(* Visualisation DALI 647/Configuration Pages/visuDALIGroups
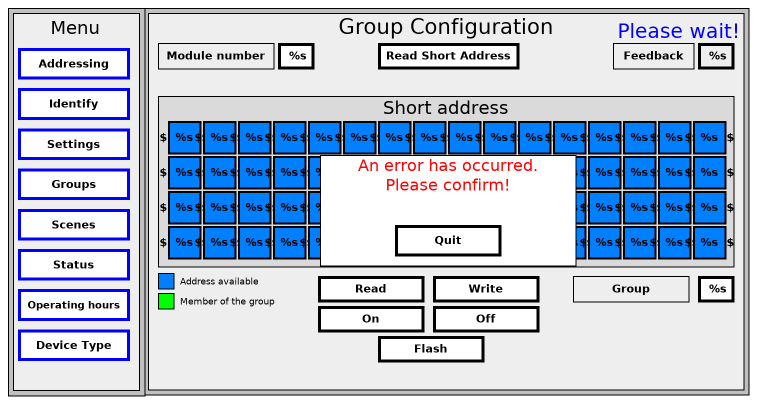
rectangle at (140,5)-(736,382): text "Group Configuration"
rectangle at (150,88)-(726,259): text "Short address"
embedded screen at (160,113)-(193,146): visuGroupButton
embedded screen at (160,148)-(193,181): visuGroupButton
embedded screen at (160,183)-(193,216): visuGroupButton
embedded screen at (160,218)-(193,251): visuGroupButton
embedded screen at (195,113)-(228,146): visuGroupButton
embedded screen at (195,148)-(228,181): visuGroupButton
embedded screen at (195,183)-(228,216): visuGroupButton
embedded screen at (195,218)-(228,251): visuGroupButton
embedded screen at (230,113)-(263,146): visuGroupButton
embedded screen at (230,148)-(263,181): visuGroupButton
embedded screen at (230,183)-(263,216): visuGroupButton
embedded screen at (230,218)-(263,251): visuGroupButton
embedded screen at (265,113)-(298,146): visuGroupButton
embedded screen at (265,148)-(298,181): visuGroupButton
embedded screen at (265,183)-(298,216): visuGroupButton
embedded screen at (265,218)-(298,251): visuGroupButton
embedded screen at (300,113)-(333,146): visuGroupButton
embedded screen at (300,148)-(333,181): visuGroupButton
embedded screen at (300,183)-(333,216): visuGroupButton
embedded screen at (300,218)-(333,251): visuGroupButton
embedded screen at (335,113)-(368,146): visuGroupButton
embedded screen at (335,148)-(368,181): visuGroupButton
embedded screen at (335,183)-(368,216): visuGroupButton
embedded screen at (335,218)-(368,251): visuGroupButton
embedded screen at (370,113)-(403,146): visuGroupButton
embedded screen at (370,148)-(403,181): visuGroupButton
embedded screen at (370,183)-(403,216): visuGroupButton
embedded screen at (370,218)-(403,251): visuGroupButton
embedded screen at (405,113)-(438,146): visuGroupButton
embedded screen at (405,148)-(438,181): visuGroupButton
embedded screen at (405,183)-(438,216): visuGroupButton
embedded screen at (405,218)-(438,251): visuGroupButton
embedded screen at (440,113)-(473,146): visuGroupButton
embedded screen at (440,148)-(473,181): visuGroupButton
embedded screen at (440,183)-(473,216): visuGroupButton
embedded screen at (440,218)-(473,251): visuGroupButton
embedded screen at (475,113)-(508,146): visuGroupButton
embedded screen at (475,148)-(508,181): visuGroupButton
embedded screen at (475,183)-(508,216): visuGroupButton
embedded screen at (475,218)-(508,251): visuGroupButton
embedded screen at (510,113)-(543,146): visuGroupButton
embedded screen at (510,148)-(543,181): visuGroupButton
embedded screen at (510,183)-(543,216): visuGroupButton
embedded screen at (510,218)-(543,251): visuGroupButton
embedded screen at (545,113)-(578,146): visuGroupButton
embedded screen at (545,148)-(578,181): visuGroupButton
embedded screen at (545,183)-(578,216): visuGroupButton
embedded screen at (545,218)-(578,251): visuGroupButton
embedded screen at (580,113)-(613,146): visuGroupButton
embedded screen at (580,148)-(613,181): visuGroupButton
embedded screen at (580,183)-(613,216): visuGroupButton
embedded screen at (580,218)-(613,251): visuGroupButton
embedded screen at (615,113)-(648,146): visuGroupButton
embedded screen at (615,148)-(648,181): visuGroupButton
embedded screen at (615,183)-(648,216): visuGroupButton
embedded screen at (615,218)-(648,251): visuGroupButton
embedded screen at (650,113)-(683,146): visuGroupButton
embedded screen at (650,148)-(683,181): visuGroupButton
embedded screen at (650,183)-(683,216): visuGroupButton
embedded screen at (650,218)-(683,251): visuGroupButton
embedded screen at (685,113)-(718,146): visuGroupButton
embedded screen at (685,148)-(718,181): visuGroupButton
embedded screen at (685,183)-(718,216): visuGroupButton
embedded screen at (685,218)-(718,251): visuGroupButton
rounded rectangle at (150,35)-(266,61): text "Module number"
rounded rectangle at (270,35)-(306,61): text "%s"; shows PrgDALIConfig.bModule_753_647; editable
rounded rectangle at (565,268)-(681,294): text "Group"
rounded rectangle at (690,268)-(726,294): text "%s"; shows PrgDALIConfig.GroupConfig.bGroup; editable
rounded rectangle at (310,268)-(416,294): text "Read"; alarm colour if PrgDALIConfig.GroupConfig.xRead; taps PrgDALIConfig.GroupConfig.xRead
rounded rectangle at (425,268)-(531,294): text "Write"; alarm colour if PrgDALIConfig.GroupConfig.xWrite; taps PrgDALIConfig.GroupConfig.xWrite
rectangle at (170,283)-(300,304): text "Member of the group"
rectangle at (170,263)-(300,284): text "Address available"
rounded rectangle at (370,328)-(476,354): text "Flash"; alarm colour if PrgDALIConfig.GroupConfig.xFlash; toggles PrgDALIConfig.GroupConfig.xFlash
rounded rectangle at (425,298)-(531,324): text "Off"; alarm colour if PrgDALIConfig.GroupConfig.xGroupOff; taps PrgDALIConfig.GroupConfig.xGroupOff
rounded rectangle at (310,298)-(416,324): text "On"; alarm colour if PrgDALIConfig.GroupConfig.xGroupOn; taps PrgDALIConfig.GroupConfig.xGroupOn
rounded rectangle at (605,35)-(686,61): text "Feedback"
rounded rectangle at (690,35)-(726,61): text "%s"; shows PrgDALIConfig.GroupConfig.bFeedback
rounded rectangle at (370,35)-(511,61): text "Read Short Address"; alarm colour if PrgDALIConfig.GroupConfig.xQueryShortAddress; taps PrgDALIConfig.GroupConfig.xQueryShortAddress
embedded screen at (0,0)-(137,388): visuDALI_Menue
group at (0,7)-(734,379)
  rectangle at (3,3)-(734,321): text "Please wait!"
group at (312,147)-(568,258)
  rectangle at (0,0)-(256,111): text "An error has occurred. / Please confirm!"
  rounded rectangle at (75,70)-(181,101): text "Quit"; taps PrgDALIConfig.GroupConfig.xQuit
4 more shapes without text or variables
*)

(* Visualisation DALI 647/Configuration Pages/visuDALIOperatingHours
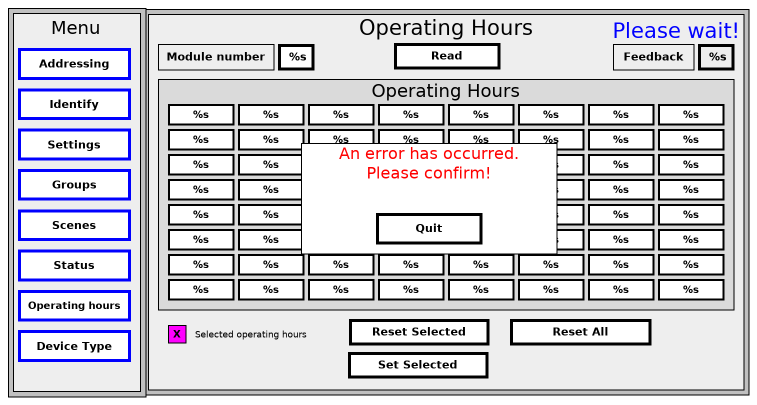
rectangle at (140,6)-(736,382): text "Operating Hours"
rectangle at (150,71)-(726,302): text "Operating Hours"
rectangle at (160,317)-(178,335): text "X"
rounded rectangle at (150,36)-(266,62): text "Module number"
rounded rectangle at (270,36)-(306,62): text "%s"; shows PrgDALIConfig.bModule_753_647; editable
rounded rectangle at (341,311)-(481,337): text "Reset Selected"; alarm colour if PrgDALIConfig.OperatingHours.xResetSelected; taps PrgDALIConfig.OperatingHours.xResetSelected
rectangle at (185,316)-(315,337): text "Selected operating hours"
rounded rectangle at (605,36)-(686,62): text "Feedback"
rounded rectangle at (690,36)-(726,62): text "%s"; shows PrgDALIConfig.OperatingHours.bFeedback
rounded rectangle at (502,311)-(643,337): text "Reset All"; alarm colour if PrgDALIConfig.OperatingHours.xResetAll; taps PrgDALIConfig.OperatingHours.xResetAll
rounded rectangle at (340,344)-(480,370): text "Set Selected"; invisible if PrgDALIConfig.OperatingHours.OldFirmware; alarm colour if PrgDALIConfig.OperatingHours.xSetSelected; taps PrgDALIConfig.OperatingHours.xSetSelected
embedded screen at (160,96)-(226,117): visuOperatingHours
embedded screen at (230,96)-(296,117): visuOperatingHours
embedded screen at (300,96)-(366,117): visuOperatingHours
embedded screen at (370,96)-(436,117): visuOperatingHours
embedded screen at (440,96)-(506,117): visuOperatingHours
embedded screen at (510,96)-(576,117): visuOperatingHours
embedded screen at (580,96)-(646,117): visuOperatingHours
embedded screen at (650,96)-(716,117): visuOperatingHours
embedded screen at (160,121)-(226,142): visuOperatingHours
embedded screen at (230,121)-(296,142): visuOperatingHours
embedded screen at (300,121)-(366,142): visuOperatingHours
embedded screen at (370,121)-(436,142): visuOperatingHours
embedded screen at (440,121)-(506,142): visuOperatingHours
embedded screen at (510,121)-(576,142): visuOperatingHours
embedded screen at (580,121)-(646,142): visuOperatingHours
embedded screen at (650,121)-(716,142): visuOperatingHours
embedded screen at (160,146)-(226,167): visuOperatingHours
embedded screen at (230,146)-(296,167): visuOperatingHours
embedded screen at (300,146)-(366,167): visuOperatingHours
embedded screen at (370,146)-(436,167): visuOperatingHours
embedded screen at (440,146)-(506,167): visuOperatingHours
embedded screen at (510,146)-(576,167): visuOperatingHours
embedded screen at (580,146)-(646,167): visuOperatingHours
embedded screen at (650,146)-(716,167): visuOperatingHours
embedded screen at (160,171)-(226,192): visuOperatingHours
embedded screen at (230,171)-(296,192): visuOperatingHours
embedded screen at (300,171)-(366,192): visuOperatingHours
embedded screen at (370,171)-(436,192): visuOperatingHours
embedded screen at (440,171)-(506,192): visuOperatingHours
embedded screen at (510,171)-(576,192): visuOperatingHours
embedded screen at (580,171)-(646,192): visuOperatingHours
embedded screen at (650,171)-(716,192): visuOperatingHours
embedded screen at (160,196)-(226,217): visuOperatingHours
embedded screen at (230,196)-(296,217): visuOperatingHours
embedded screen at (300,196)-(366,217): visuOperatingHours
embedded screen at (370,196)-(436,217): visuOperatingHours
embedded screen at (440,196)-(506,217): visuOperatingHours
embedded screen at (510,196)-(576,217): visuOperatingHours
embedded screen at (580,196)-(646,217): visuOperatingHours
embedded screen at (650,196)-(716,217): visuOperatingHours
embedded screen at (160,221)-(226,242): visuOperatingHours
embedded screen at (230,221)-(296,242): visuOperatingHours
embedded screen at (300,221)-(366,242): visuOperatingHours
embedded screen at (370,221)-(436,242): visuOperatingHours
embedded screen at (440,221)-(506,242): visuOperatingHours
embedded screen at (510,221)-(576,242): visuOperatingHours
embedded screen at (580,221)-(646,242): visuOperatingHours
embedded screen at (650,221)-(716,242): visuOperatingHours
embedded screen at (160,246)-(226,267): visuOperatingHours
embedded screen at (230,246)-(296,267): visuOperatingHours
embedded screen at (300,246)-(366,267): visuOperatingHours
embedded screen at (370,246)-(436,267): visuOperatingHours
embedded screen at (440,246)-(506,267): visuOperatingHours
embedded screen at (510,246)-(576,267): visuOperatingHours
embedded screen at (580,246)-(646,267): visuOperatingHours
embedded screen at (650,246)-(716,267): visuOperatingHours
embedded screen at (160,271)-(226,292): visuOperatingHours
embedded screen at (230,271)-(296,292): visuOperatingHours
embedded screen at (300,271)-(366,292): visuOperatingHours
embedded screen at (370,271)-(436,292): visuOperatingHours
embedded screen at (440,271)-(506,292): visuOperatingHours
embedded screen at (510,271)-(576,292): visuOperatingHours
embedded screen at (580,271)-(646,292): visuOperatingHours
embedded screen at (650,271)-(716,292): visuOperatingHours
rounded rectangle at (386,35)-(492,61): text "Read"; alarm colour if PrgDALIConfig.OperatingHours.xEnable; taps PrgDALIConfig.OperatingHours.xEnable
embedded screen at (0,0)-(138,389): visuDALI_Menue
rectangle at (3,9)-(734,383): text "Please wait!"; invisible if PrgDALIConfig.OperatingHours.xReady
group at (293,135)-(549,246)
  rectangle at (0,0)-(256,111): text "An error has occurred. / Please confirm!"
  rounded rectangle at (75,70)-(181,101): text "Quit"; taps PrgDALIConfig.OperatingHours.xQuit
1 more shapes without text or variables
*)

(* Visualisation DALI 647/Configuration Pages/visuDALIScenes
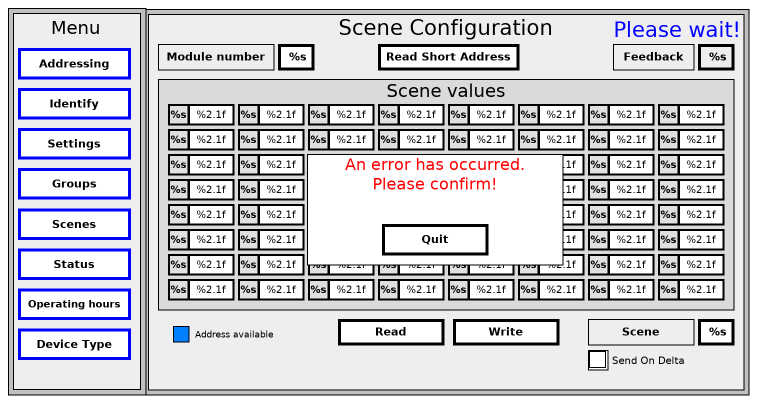
rectangle at (140,6)-(736,382): text "Scene Configuration"
rectangle at (150,71)-(726,302): text "Scene values"
rounded rectangle at (150,36)-(266,62): text "Module number"
rounded rectangle at (270,36)-(306,62): text "%s"; shows PrgDALIConfig.bModule_753_647; editable
rounded rectangle at (330,311)-(436,337): text "Read"; alarm colour if PrgDALIConfig.SceneConfig.xRead; taps PrgDALIConfig.SceneConfig.xRead
rounded rectangle at (445,311)-(551,337): text "Write"; alarm colour if PrgDALIConfig.SceneConfig.xWrite; taps PrgDALIConfig.SceneConfig.xWrite
rectangle at (185,316)-(281,337): text "Address available"
rounded rectangle at (605,36)-(686,62): text "Feedback"
rounded rectangle at (690,36)-(726,62): text "%s"; shows PrgDALIConfig.SceneConfig.bFeedback
rounded rectangle at (370,36)-(511,62): text "Read Short Address"; alarm colour if PrgDALIConfig.SceneConfig.xQueryShortAddress; taps PrgDALIConfig.SceneConfig.xQueryShortAddress
embedded screen at (580,342)-(600,362): visuDaliSelect
embedded screen at (160,96)-(226,117): visuSceneValues
embedded screen at (230,96)-(296,117): visuSceneValues
embedded screen at (300,96)-(366,117): visuSceneValues
embedded screen at (370,96)-(436,117): visuSceneValues
embedded screen at (440,96)-(506,117): visuSceneValues
embedded screen at (510,96)-(576,117): visuSceneValues
embedded screen at (580,96)-(646,117): visuSceneValues
embedded screen at (650,96)-(716,117): visuSceneValues
embedded screen at (160,121)-(226,142): visuSceneValues
embedded screen at (230,121)-(296,142): visuSceneValues
embedded screen at (300,121)-(366,142): visuSceneValues
embedded screen at (370,121)-(436,142): visuSceneValues
embedded screen at (440,121)-(506,142): visuSceneValues
embedded screen at (510,121)-(576,142): visuSceneValues
embedded screen at (580,121)-(646,142): visuSceneValues
embedded screen at (650,121)-(716,142): visuSceneValues
embedded screen at (160,146)-(226,167): visuSceneValues
embedded screen at (230,146)-(296,167): visuSceneValues
embedded screen at (300,146)-(366,167): visuSceneValues
embedded screen at (370,146)-(436,167): visuSceneValues
embedded screen at (440,146)-(506,167): visuSceneValues
embedded screen at (510,146)-(576,167): visuSceneValues
embedded screen at (580,146)-(646,167): visuSceneValues
embedded screen at (650,146)-(716,167): visuSceneValues
embedded screen at (160,171)-(226,192): visuSceneValues
embedded screen at (230,171)-(296,192): visuSceneValues
embedded screen at (300,171)-(366,192): visuSceneValues
embedded screen at (370,171)-(436,192): visuSceneValues
embedded screen at (440,171)-(506,192): visuSceneValues
embedded screen at (510,171)-(576,192): visuSceneValues
embedded screen at (580,171)-(646,192): visuSceneValues
embedded screen at (650,171)-(716,192): visuSceneValues
embedded screen at (160,196)-(226,217): visuSceneValues
embedded screen at (230,196)-(296,217): visuSceneValues
embedded screen at (300,196)-(366,217): visuSceneValues
embedded screen at (370,196)-(436,217): visuSceneValues
embedded screen at (440,196)-(506,217): visuSceneValues
embedded screen at (510,196)-(576,217): visuSceneValues
embedded screen at (580,196)-(646,217): visuSceneValues
embedded screen at (650,196)-(716,217): visuSceneValues
embedded screen at (160,221)-(226,242): visuSceneValues
embedded screen at (230,221)-(296,242): visuSceneValues
embedded screen at (300,221)-(366,242): visuSceneValues
embedded screen at (370,221)-(436,242): visuSceneValues
embedded screen at (440,221)-(506,242): visuSceneValues
embedded screen at (510,221)-(576,242): visuSceneValues
embedded screen at (580,221)-(646,242): visuSceneValues
embedded screen at (650,221)-(716,242): visuSceneValues
embedded screen at (160,246)-(226,267): visuSceneValues
embedded screen at (230,246)-(296,267): visuSceneValues
embedded screen at (300,246)-(366,267): visuSceneValues
embedded screen at (370,246)-(436,267): visuSceneValues
embedded screen at (440,246)-(506,267): visuSceneValues
embedded screen at (510,246)-(576,267): visuSceneValues
embedded screen at (580,246)-(646,267): visuSceneValues
embedded screen at (650,246)-(716,267): visuSceneValues
embedded screen at (160,271)-(226,292): visuSceneValues
embedded screen at (230,271)-(296,292): visuSceneValues
embedded screen at (300,271)-(366,292): visuSceneValues
embedded screen at (370,271)-(436,292): visuSceneValues
embedded screen at (440,271)-(506,292): visuSceneValues
embedded screen at (510,271)-(576,292): visuSceneValues
embedded screen at (580,271)-(646,292): visuSceneValues
embedded screen at (650,271)-(716,292): visuSceneValues
rounded rectangle at (580,311)-(686,337): text "Scene"
rounded rectangle at (690,311)-(726,337): text "%s"; shows PrgDALIConfig.SceneConfig.bScene; editable
embedded screen at (0,0)-(138,387): visuDALI_Menue
rectangle at (4,8)-(735,381): text "Please wait!"; invisible if PrgDALIConfig.SceneConfig.xReady
group at (299,146)-(555,257)
  rectangle at (0,0)-(256,111): text "An error has occurred. / Please confirm!"
  rounded rectangle at (75,70)-(181,101): text "Quit"; taps PrgDALIConfig.SceneConfig.xQuit
rectangle at (602,341)-(690,364): text "Send On Delta"
2 more shapes without text or variables
*)

(* Visualisation DALI 647/Private/visuDaliSelect
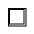
rectangle at (1,1)-(16,16): invisible if $Select$; toggles $Select$
2 more shapes without text or variables
*)

(* Visualisation Private/English/visuECG_settings
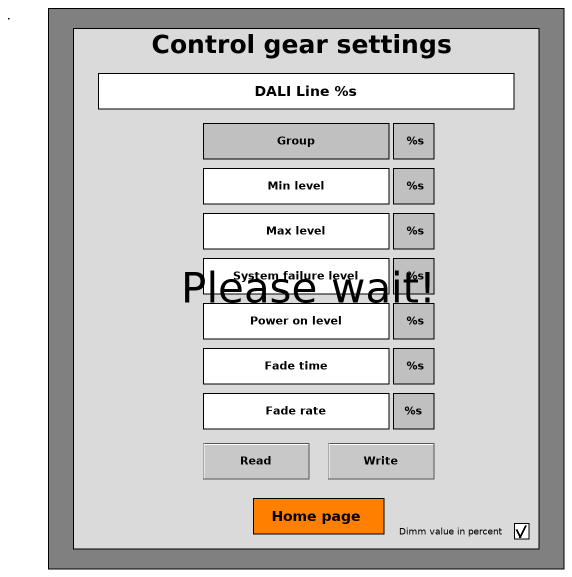
rectangle at (150,40)-(616,561): text "Control gear settings"
rectangle at (280,225)-(466,261): text "Max level"
rectangle at (280,180)-(466,216): text "Min level"
rectangle at (280,270)-(466,306): text "System failure level"
rectangle at (280,315)-(466,351): text "Power on level"
rectangle at (280,360)-(466,396): text "Fade time"
rectangle at (280,405)-(466,441): text "Fade rate"
rectangle at (280,135)-(466,171): text "Short address"; invisible if DALI_Config.Kurzadr_Gruppe; toggles DALI_Config.Kurzadr_Gruppe
rectangle at (280,135)-(466,171): text "Group"; invisible if not DALI_Config.Kurzadr_Gruppe; toggles DALI_Config.Kurzadr_Gruppe; tooltip Selection group or short address
rectangle at (470,135)-(511,171): text "%s"; shows DALI_Config.Adresse; tooltip Enter group (1-16) or short address (1 - 64); editable
rounded rectangle at (330,510)-(461,546): text "Home page"; opens visuFrontPageDALI; tooltip Back to home page
rectangle at (470,180)-(511,216): text "%s"; shows DALI_Config.MinLevel; tooltip Minimal brightness level in percent. Min level has to be smaller than max level.; editable
rectangle at (470,225)-(511,261): text "%s"; shows DALI_Config.MaxLevel; tooltip Maximum brightness level in percent; editable
rectangle at (470,270)-(511,306): text "%s"; shows DALI_Config.SystemFailure; tooltip Brightness level in percent in case of a system failure. The value 101 means "MASK".; editable
rectangle at (470,315)-(511,351): text "%s"; shows DALI_Config.PowerOn; tooltip Brightness level in percent if the ECGs are powered on.; editable
rectangle at (470,360)-(511,396): text "%s"; shows DALI_Config.Konfig[4]; tooltip Enter the fade time (0 - 15); editable
rectangle at (470,405)-(511,441): text "%s"; shows DALI_Config.Konfig[5]; tooltip Enter the fade rate (1 -15); editable
button at (280,455)-(386,491): text "Read"; taps DALI_Config.Lese; tooltip If you click the button "Read", the settings of the ECG will be read. Group queries are not possible.
button at (405,455)-(511,491): text "Write"; taps DALI_Config.Schreib; tooltip If you click the button "Write", the new settings will be written into the ECG.
rounded rectangle at (175,85)-(591,121): text "DALI Line %s"; shows DALI_Config.Dali_Linie; alarm colour if DALI_Config.keineJobliste; tooltip You can change the DALI Line only on the home page.
rectangle at (474,532)-(590,555): text "Dimm value in percent"
rectangle at (591,535)-(606,551): toggles DALI_Config.xDimmwertProzent
polyline at (593,537)-(603,549): invisible if NOT  DALI_Config.xDimmwertProzent; toggles DALI_Config.xDimmwertProzent
rectangle at (153,101)-(618,498): text "Please wait!"; invisible if NOT DALI_Config.JobMerker[16] AND NOT DALI_Config.JobMerker[11]
2 more shapes without text or variables
*)

(* Visualisation visuFrontPageDALI
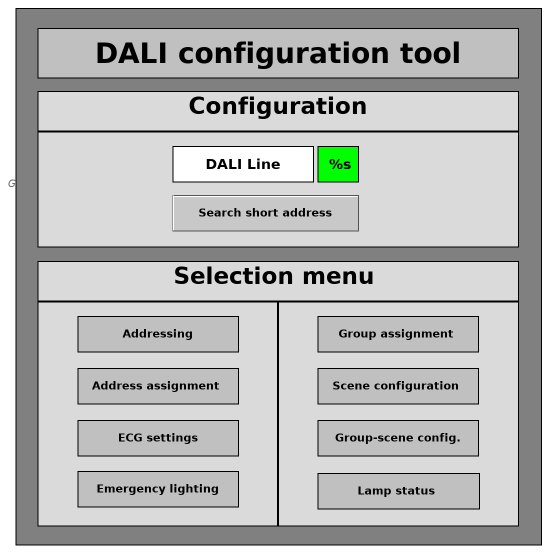
embedded screen at (178,137)-(206,164): Addressing
embedded screen at (211,137)-(239,165): ECG_settings
embedded screen at (214,173)-(235,196): GroupSceneConfiguration
embedded screen at (179,171)-(198,196): Group_assignment
embedded screen at (177,200)-(198,224): Lamp_status
embedded screen at (209,200)-(230,223): Scene_configuration
embedded screen at (236,198)-(260,218): Sort_short_address
rectangle at (171,91)-(652,247): text "Configuration"
rectangle at (171,261)-(652,526): text "Selection menu"
rectangle at (171,28)-(652,78): text "DALI configuration tool"
rectangle at (211,316)-(372,352): text "Addressing"; opens visuAddressing
rectangle at (211,368)-(372,404): text "Address assignment"; opens visuSort_short_address
rectangle at (451,316)-(612,352): text "Group assignment"; opens visugroup_assignment
rectangle at (451,368)-(612,404): text "Scene configuration"; opens visuScene_configuration
rectangle at (211,420)-(372,456): text "ECG settings"; opens visuECG_settings
rectangle at (451,420)-(612,456): text "Group-scene config."; opens visuGroupSceneConfiguration
rectangle at (306,146)-(447,182): text "DALI Line"
button at (306,195)-(492,231): text "Search short address"; taps DALI_Config.SucheKurzadr; tooltip Clicking the button "Search Short Address" will start the search for available short addresses.
rectangle at (451,146)-(492,182): text "%s"; shows DALI_Config.Dali_Linie; alarm colour if DALI_Config.keineJobliste; tooltip Select DALI Line (1 - 5); editable
rectangle at (451,473)-(613,509): text "Lamp status"; opens visuLamp_status
rectangle at (211,471)-(372,507): text "Emergency lighting"; invisible if NOT .EmergencyLighting; opens visuConfigurationEmergencyLighting
4 more shapes without text or variables
*)

(* Visualisation Private/English/visuGroup_assignment
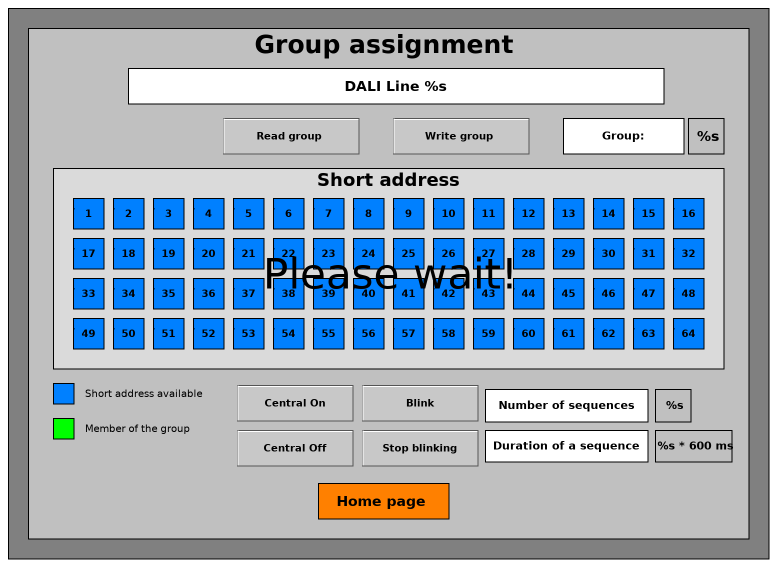
rectangle at (40,40)-(761,551): text "Group assignment"
rounded rectangle at (330,495)-(461,531): text "Home page"; opens visuFrontPageDALI; tooltip Back to home page
rectangle at (65,180)-(736,381): text "Short address"
rectangle at (85,210)-(116,241): text "1"; alarm colour if DALI_Config.Kurzadr[1]
rectangle at (85,210)-(116,241): text "1"; invisible if not DALI_Config.Kurzadr[1]; alarm colour if DALI_Config.Gruppenadr[1]; toggles DALI_Config.Gruppenadr[1]
rectangle at (125,210)-(156,241): text "2"; alarm colour if DALI_Config.Kurzadr[2]
rectangle at (125,210)-(156,241): text "2"; invisible if not DALI_Config.Kurzadr[2]; alarm colour if DALI_Config.Gruppenadr[2]; toggles DALI_Config.Gruppenadr[2]
rectangle at (165,210)-(196,241): text "3"; alarm colour if DALI_Config.Kurzadr[3]
rectangle at (165,210)-(196,241): text "3"; invisible if not DALI_Config.Kurzadr[3]; alarm colour if DALI_Config.Gruppenadr[3]; toggles DALI_Config.Gruppenadr[3]
rectangle at (205,210)-(236,241): text "4"; alarm colour if DALI_Config.Kurzadr[4]
rectangle at (205,210)-(236,241): text "4"; invisible if not DALI_Config.Kurzadr[4]; alarm colour if DALI_Config.Gruppenadr[4]; toggles DALI_Config.Gruppenadr[4]
rectangle at (245,210)-(276,241): text "5"; alarm colour if DALI_Config.Kurzadr[5]
rectangle at (245,210)-(276,241): text "5"; invisible if not DALI_Config.Kurzadr[5]; alarm colour if DALI_Config.Gruppenadr[5]; toggles DALI_Config.Gruppenadr[5]
rectangle at (285,210)-(316,241): text "6"; alarm colour if DALI_Config.Kurzadr[6]
rectangle at (285,210)-(316,241): text "6"; invisible if not DALI_Config.Kurzadr[6]; alarm colour if DALI_Config.Gruppenadr[6]; toggles DALI_Config.Gruppenadr[6]
rectangle at (325,210)-(356,241): text "7"; alarm colour if DALI_Config.Kurzadr[7]
rectangle at (325,210)-(356,241): text "7"; invisible if not DALI_Config.Kurzadr[7]; alarm colour if DALI_Config.Gruppenadr[7]; toggles DALI_Config.Gruppenadr[7]
rectangle at (365,210)-(396,241): text "8"; alarm colour if DALI_Config.Kurzadr[8]
rectangle at (365,210)-(396,241): text "8"; invisible if not DALI_Config.Kurzadr[8]; alarm colour if DALI_Config.Gruppenadr[8]; toggles DALI_Config.Gruppenadr[8]
rectangle at (405,210)-(436,241): text "9"; alarm colour if DALI_Config.Kurzadr[9]
rectangle at (405,210)-(436,241): text "9"; invisible if not DALI_Config.Kurzadr[9]; alarm colour if DALI_Config.Gruppenadr[9]; toggles DALI_Config.Gruppenadr[9]
rectangle at (445,210)-(476,241): text "10"; alarm colour if DALI_Config.Kurzadr[10]
rectangle at (445,210)-(476,241): text "10"; invisible if not DALI_Config.Kurzadr[10]; alarm colour if DALI_Config.Gruppenadr[10]; toggles DALI_Config.Gruppenadr[10]
rectangle at (485,210)-(516,241): text "11"; alarm colour if DALI_Config.Kurzadr[11]
rectangle at (485,210)-(516,241): text "11"; invisible if not DALI_Config.Kurzadr[11]; alarm colour if DALI_Config.Gruppenadr[11]; toggles DALI_Config.Gruppenadr[11]
rectangle at (525,210)-(556,241): text "12"; alarm colour if DALI_Config.Kurzadr[12]
rectangle at (525,210)-(556,241): text "12"; invisible if not DALI_Config.Kurzadr[12]; alarm colour if DALI_Config.Gruppenadr[12]; toggles DALI_Config.Gruppenadr[12]
rectangle at (565,210)-(596,241): text "13"; alarm colour if DALI_Config.Kurzadr[13]
rectangle at (565,210)-(596,241): text "13"; invisible if not DALI_Config.Kurzadr[13]; alarm colour if DALI_Config.Gruppenadr[13]; toggles DALI_Config.Gruppenadr[13]
rectangle at (605,210)-(636,241): text "14"; alarm colour if DALI_Config.Kurzadr[14]
rectangle at (605,210)-(636,241): text "14"; invisible if not DALI_Config.Kurzadr[14]; alarm colour if DALI_Config.Gruppenadr[14]; toggles DALI_Config.Gruppenadr[14]
rectangle at (645,210)-(676,241): text "15"; alarm colour if DALI_Config.Kurzadr[15]
rectangle at (645,210)-(676,241): text "15"; invisible if not DALI_Config.Kurzadr[15]; alarm colour if DALI_Config.Gruppenadr[15]; toggles DALI_Config.Gruppenadr[15]
rectangle at (685,210)-(716,241): text "16"; alarm colour if DALI_Config.Kurzadr[16]
rectangle at (685,210)-(716,241): text "16"; invisible if not DALI_Config.Kurzadr[16]; alarm colour if DALI_Config.Gruppenadr[16]; toggles DALI_Config.Gruppenadr[16]
button at (405,130)-(541,166): text "Write group"; taps DALI_Config.Gruppenkonfiguration; tooltip If you click the button "Write Group", the marked short addresses will be saved as a group.
rectangle at (575,130)-(696,166): text "Group:"
rectangle at (700,130)-(736,166): text "%s"; shows DALI_Config.Gruppe; tooltip Enter the number of the group (1 - 16); editable
button at (235,130)-(371,166): text "Read group"; taps DALI_Config.GruppeLesen; tooltip If you click the button "Read Group", the short addresses that belong to the group will be displayed.
rectangle at (95,395)-(226,416): text "Short address available"
rectangle at (95,430)-(246,451): text "Member of the group"
rounded rectangle at (140,80)-(676,116): text "DALI Line %s"; shows DALI_Config.Dali_Linie; alarm colour if DALI_Config.keineJobliste; tooltip You can change the DALI Line only on the home page.
rectangle at (85,250)-(116,281): text "17"; alarm colour if DALI_Config.Kurzadr[17]
rectangle at (85,250)-(116,281): text "17"; invisible if not DALI_Config.Kurzadr[17]; alarm colour if DALI_Config.Gruppenadr[17]; toggles DALI_Config.Gruppenadr[17]
rectangle at (125,250)-(156,281): text "18"; alarm colour if DALI_Config.Kurzadr[18]
rectangle at (125,250)-(156,281): text "18"; invisible if not DALI_Config.Kurzadr[18]; alarm colour if DALI_Config.Gruppenadr[18]; toggles DALI_Config.Gruppenadr[18]
rectangle at (165,250)-(196,281): text "19"; alarm colour if DALI_Config.Kurzadr[19]
rectangle at (165,250)-(196,281): text "19"; invisible if not DALI_Config.Kurzadr[19]; alarm colour if DALI_Config.Gruppenadr[19]; toggles DALI_Config.Gruppenadr[19]
rectangle at (205,250)-(236,281): text "20"; alarm colour if DALI_Config.Kurzadr[20]
rectangle at (205,250)-(236,281): text "20"; invisible if not DALI_Config.Kurzadr[20]; alarm colour if DALI_Config.Gruppenadr[20]; toggles DALI_Config.Gruppenadr[20]
rectangle at (245,250)-(276,281): text "21"; alarm colour if DALI_Config.Kurzadr[21]
rectangle at (245,250)-(276,281): text "21"; invisible if not DALI_Config.Kurzadr[21]; alarm colour if DALI_Config.Gruppenadr[21]; toggles DALI_Config.Gruppenadr[21]
rectangle at (285,250)-(316,281): text "22"; alarm colour if DALI_Config.Kurzadr[22]
rectangle at (285,250)-(316,281): text "22"; invisible if not DALI_Config.Kurzadr[22]; alarm colour if DALI_Config.Gruppenadr[22]; toggles DALI_Config.Gruppenadr[22]
rectangle at (325,250)-(356,281): text "23"; alarm colour if DALI_Config.Kurzadr[23]
rectangle at (325,250)-(356,281): text "23"; invisible if not DALI_Config.Kurzadr[23]; alarm colour if DALI_Config.Gruppenadr[23]; toggles DALI_Config.Gruppenadr[23]
rectangle at (365,250)-(396,281): text "24"; alarm colour if DALI_Config.Kurzadr[24]
rectangle at (365,250)-(396,281): text "24"; invisible if not DALI_Config.Kurzadr[24]; alarm colour if DALI_Config.Gruppenadr[24]; toggles DALI_Config.Gruppenadr[24]
rectangle at (405,250)-(436,281): text "25"; alarm colour if DALI_Config.Kurzadr[25]
rectangle at (405,250)-(436,281): text "25"; invisible if not DALI_Config.Kurzadr[25]; alarm colour if DALI_Config.Gruppenadr[25]; toggles DALI_Config.Gruppenadr[25]
rectangle at (445,250)-(476,281): text "26"; alarm colour if DALI_Config.Kurzadr[26]
rectangle at (445,250)-(476,281): text "26"; invisible if not DALI_Config.Kurzadr[26]; alarm colour if DALI_Config.Gruppenadr[26]; toggles DALI_Config.Gruppenadr[26]
rectangle at (485,250)-(516,281): text "27"; alarm colour if DALI_Config.Kurzadr[27]
rectangle at (485,250)-(516,281): text "27"; invisible if not DALI_Config.Kurzadr[27]; alarm colour if DALI_Config.Gruppenadr[27]; toggles DALI_Config.Gruppenadr[27]
rectangle at (525,250)-(556,281): text "28"; alarm colour if DALI_Config.Kurzadr[28]
rectangle at (525,250)-(556,281): text "28"; invisible if not DALI_Config.Kurzadr[28]; alarm colour if DALI_Config.Gruppenadr[28]; toggles DALI_Config.Gruppenadr[28]
rectangle at (565,250)-(596,281): text "29"; alarm colour if DALI_Config.Kurzadr[29]
rectangle at (565,250)-(596,281): text "29"; invisible if not DALI_Config.Kurzadr[29]; alarm colour if DALI_Config.Gruppenadr[29]; toggles DALI_Config.Gruppenadr[29]
rectangle at (605,250)-(636,281): text "30"; alarm colour if DALI_Config.Kurzadr[30]
rectangle at (605,250)-(636,281): text "30"; invisible if not DALI_Config.Kurzadr[30]; alarm colour if DALI_Config.Gruppenadr[30]; toggles DALI_Config.Gruppenadr[30]
rectangle at (645,250)-(676,281): text "31"; alarm colour if DALI_Config.Kurzadr[31]
rectangle at (645,250)-(676,281): text "31"; invisible if not DALI_Config.Kurzadr[31]; alarm colour if DALI_Config.Gruppenadr[31]; toggles DALI_Config.Gruppenadr[31]
rectangle at (685,250)-(716,281): text "32"; alarm colour if DALI_Config.Kurzadr[32]
rectangle at (685,250)-(716,281): text "32"; invisible if not DALI_Config.Kurzadr[32]; alarm colour if DALI_Config.Gruppenadr[32]; toggles DALI_Config.Gruppenadr[32]
rectangle at (85,290)-(116,321): text "33"; alarm colour if DALI_Config.Kurzadr[33]
rectangle at (85,290)-(116,321): text "33"; invisible if not DALI_Config.Kurzadr[33]; alarm colour if DALI_Config.Gruppenadr[33]; toggles DALI_Config.Gruppenadr[33]
rectangle at (125,290)-(156,321): text "34"; alarm colour if DALI_Config.Kurzadr[34]
rectangle at (125,290)-(156,321): text "34"; invisible if not DALI_Config.Kurzadr[34]; alarm colour if DALI_Config.Gruppenadr[34]; toggles DALI_Config.Gruppenadr[34]
rectangle at (165,290)-(196,321): text "35"; alarm colour if DALI_Config.Kurzadr[35]
rectangle at (165,290)-(196,321): text "35"; invisible if not DALI_Config.Kurzadr[35]; alarm colour if DALI_Config.Gruppenadr[35]; toggles DALI_Config.Gruppenadr[35]
rectangle at (205,290)-(236,321): text "36"; alarm colour if DALI_Config.Kurzadr[36]
rectangle at (205,290)-(236,321): text "36"; invisible if not DALI_Config.Kurzadr[36]; alarm colour if DALI_Config.Gruppenadr[36]; toggles DALI_Config.Gruppenadr[36]
rectangle at (245,290)-(276,321): text "37"; alarm colour if DALI_Config.Kurzadr[37]
rectangle at (245,290)-(276,321): text "37"; invisible if not DALI_Config.Kurzadr[37]; alarm colour if DALI_Config.Gruppenadr[37]; toggles DALI_Config.Gruppenadr[37]
rectangle at (285,290)-(316,321): text "38"; alarm colour if DALI_Config.Kurzadr[38]
rectangle at (285,290)-(316,321): text "38"; invisible if not DALI_Config.Kurzadr[38]; alarm colour if DALI_Config.Gruppenadr[38]; toggles DALI_Config.Gruppenadr[38]
rectangle at (325,290)-(356,321): text "39"; alarm colour if DALI_Config.Kurzadr[39]
rectangle at (325,290)-(356,321): text "39"; invisible if not DALI_Config.Kurzadr[39]; alarm colour if DALI_Config.Gruppenadr[39]; toggles DALI_Config.Gruppenadr[39]
rectangle at (365,290)-(396,321): text "40"; alarm colour if DALI_Config.Kurzadr[40]
rectangle at (365,290)-(396,321): text "40"; invisible if not DALI_Config.Kurzadr[40]; alarm colour if DALI_Config.Gruppenadr[40]; toggles DALI_Config.Gruppenadr[40]
rectangle at (405,290)-(436,321): text "41"; alarm colour if DALI_Config.Kurzadr[41]
rectangle at (405,290)-(436,321): text "41"; invisible if not DALI_Config.Kurzadr[41]; alarm colour if DALI_Config.Gruppenadr[41]; toggles DALI_Config.Gruppenadr[41]
rectangle at (445,290)-(476,321): text "42"; alarm colour if DALI_Config.Kurzadr[42]
rectangle at (445,290)-(476,321): text "42"; invisible if not DALI_Config.Kurzadr[42]; alarm colour if DALI_Config.Gruppenadr[42]; toggles DALI_Config.Gruppenadr[42]
rectangle at (485,290)-(516,321): text "43"; alarm colour if DALI_Config.Kurzadr[43]
rectangle at (485,290)-(516,321): text "43"; invisible if not DALI_Config.Kurzadr[43]; alarm colour if DALI_Config.Gruppenadr[43]; toggles DALI_Config.Gruppenadr[43]
rectangle at (525,290)-(556,321): text "44"; alarm colour if DALI_Config.Kurzadr[44]
rectangle at (525,290)-(556,321): text "44"; invisible if not DALI_Config.Kurzadr[44]; alarm colour if DALI_Config.Gruppenadr[44]; toggles DALI_Config.Gruppenadr[44]
rectangle at (565,290)-(596,321): text "45"; alarm colour if DALI_Config.Kurzadr[45]
rectangle at (565,290)-(596,321): text "45"; invisible if not DALI_Config.Kurzadr[45]; alarm colour if DALI_Config.Gruppenadr[45]; toggles DALI_Config.Gruppenadr[45]
rectangle at (605,290)-(636,321): text "46"; alarm colour if DALI_Config.Kurzadr[46]
rectangle at (605,290)-(636,321): text "46"; invisible if not DALI_Config.Kurzadr[46]; alarm colour if DALI_Config.Gruppenadr[46]; toggles DALI_Config.Gruppenadr[46]
rectangle at (645,290)-(676,321): text "47"; alarm colour if DALI_Config.Kurzadr[47]
rectangle at (645,290)-(676,321): text "47"; invisible if not DALI_Config.Kurzadr[47]; alarm colour if DALI_Config.Gruppenadr[47]; toggles DALI_Config.Gruppenadr[47]
rectangle at (685,290)-(716,321): text "48"; alarm colour if DALI_Config.Kurzadr[48]
rectangle at (685,290)-(716,321): text "48"; invisible if not DALI_Config.Kurzadr[48]; alarm colour if DALI_Config.Gruppenadr[48]; toggles DALI_Config.Gruppenadr[48]
rectangle at (85,330)-(116,361): text "49"; alarm colour if DALI_Config.Kurzadr[49]
rectangle at (85,330)-(116,361): text "49"; invisible if not DALI_Config.Kurzadr[49]; alarm colour if DALI_Config.Gruppenadr[49]; toggles DALI_Config.Gruppenadr[49]
rectangle at (125,330)-(156,361): text "50"; alarm colour if DALI_Config.Kurzadr[50]
rectangle at (125,330)-(156,361): text "50"; invisible if not DALI_Config.Kurzadr[50]; alarm colour if DALI_Config.Gruppenadr[50]; toggles DALI_Config.Gruppenadr[50]
rectangle at (165,330)-(196,361): text "51"; alarm colour if DALI_Config.Kurzadr[51]
rectangle at (165,330)-(196,361): text "51"; invisible if not DALI_Config.Kurzadr[51]; alarm colour if DALI_Config.Gruppenadr[51]; toggles DALI_Config.Gruppenadr[51]
rectangle at (205,330)-(236,361): text "52"; alarm colour if DALI_Config.Kurzadr[52]
rectangle at (205,330)-(236,361): text "52"; invisible if not DALI_Config.Kurzadr[52]; alarm colour if DALI_Config.Gruppenadr[52]; toggles DALI_Config.Gruppenadr[52]
rectangle at (245,330)-(276,361): text "53"; alarm colour if DALI_Config.Kurzadr[53]
rectangle at (245,330)-(276,361): text "53"; invisible if not DALI_Config.Kurzadr[53]; alarm colour if DALI_Config.Gruppenadr[53]; toggles DALI_Config.Gruppenadr[53]
rectangle at (285,330)-(316,361): text "54"; alarm colour if DALI_Config.Kurzadr[54]
rectangle at (285,330)-(316,361): text "54"; invisible if not DALI_Config.Kurzadr[54]; alarm colour if DALI_Config.Gruppenadr[54]; toggles DALI_Config.Gruppenadr[54]
rectangle at (325,330)-(356,361): text "55"; alarm colour if DALI_Config.Kurzadr[55]
rectangle at (325,330)-(356,361): text "55"; invisible if not DALI_Config.Kurzadr[55]; alarm colour if DALI_Config.Gruppenadr[55]; toggles DALI_Config.Gruppenadr[55]
rectangle at (365,330)-(396,361): text "56"; alarm colour if DALI_Config.Kurzadr[56]
rectangle at (365,330)-(396,361): text "56"; invisible if not DALI_Config.Kurzadr[56]; alarm colour if DALI_Config.Gruppenadr[56]; toggles DALI_Config.Gruppenadr[56]
rectangle at (405,330)-(436,361): text "57"; alarm colour if DALI_Config.Kurzadr[57]
rectangle at (405,330)-(436,361): text "57"; invisible if not DALI_Config.Kurzadr[57]; alarm colour if DALI_Config.Gruppenadr[57]; toggles DALI_Config.Gruppenadr[57]
rectangle at (445,330)-(476,361): text "58"; alarm colour if DALI_Config.Kurzadr[58]
rectangle at (445,330)-(476,361): text "58"; invisible if not DALI_Config.Kurzadr[58]; alarm colour if DALI_Config.Gruppenadr[58]; toggles DALI_Config.Gruppenadr[58]
rectangle at (485,330)-(516,361): text "59"; alarm colour if DALI_Config.Kurzadr[59]
rectangle at (485,330)-(516,361): text "59"; invisible if not DALI_Config.Kurzadr[59]; alarm colour if DALI_Config.Gruppenadr[59]; toggles DALI_Config.Gruppenadr[59]
rectangle at (525,330)-(556,361): text "60"; alarm colour if DALI_Config.Kurzadr[60]
rectangle at (525,330)-(556,361): text "60"; invisible if not DALI_Config.Kurzadr[60]; alarm colour if DALI_Config.Gruppenadr[60]; toggles DALI_Config.Gruppenadr[60]
rectangle at (565,330)-(596,361): text "61"; alarm colour if DALI_Config.Kurzadr[61]
rectangle at (565,330)-(596,361): text "61"; invisible if not DALI_Config.Kurzadr[61]; alarm colour if DALI_Config.Gruppenadr[61]; toggles DALI_Config.Gruppenadr[61]
rectangle at (605,330)-(636,361): text "62"; alarm colour if DALI_Config.Kurzadr[62]
rectangle at (605,330)-(636,361): text "62"; invisible if not DALI_Config.Kurzadr[62]; alarm colour if DALI_Config.Gruppenadr[62]; toggles DALI_Config.Gruppenadr[62]
rectangle at (645,330)-(676,361): text "63"; alarm colour if DALI_Config.Kurzadr[63]
rectangle at (645,330)-(676,361): text "63"; invisible if not DALI_Config.Kurzadr[63]; alarm colour if DALI_Config.Gruppenadr[63]; toggles DALI_Config.Gruppenadr[63]
rectangle at (685,330)-(716,361): text "64"; alarm colour if DALI_Config.Kurzadr[64]
rectangle at (685,330)-(716,361): text "64"; invisible if not DALI_Config.Kurzadr[64]; alarm colour if DALI_Config.Gruppenadr[64]; toggles DALI_Config.Gruppenadr[64]
rectangle at (42,39)-(763,532): text "Please wait!"; invisible if NOT DALI_Config.Unsichtbar
button at (374,397)-(490,433): text "Blink"; taps DALI_Config.BlinkenGruppe; tooltip Über den Button "Blinken" blinkt die ausgewählte Gruppe so lange, wie es beim Parameter "Blinkzeit" eingestellt ist.
button at (374,442)-(490,478): text "Stop blinking"; taps DALI_Config.xBlinken_Aus; tooltip Über den Button "Blinken beenden" wird das Blinken der Gruppe sofort abgebrochen.
rectangle at (539,401)-(655,434): text "Blink time [sek]"; invisible if DALI_Config.bActualFirmware < 7
button at (249,442)-(365,478): text "Central Off"; taps DALI_Config.Aus; tooltip Über den Button "Zentral AUS" werden alle Leuchten ausgeschaltet.
button at (249,397)-(365,433): text "Central On"; taps DALI_Config.Ein; tooltip Über den Button "Zentral EIN" werden alle Leuchten eingeschaltet.
rectangle at (667,401)-(703,434): text "%s"; shows DALI_Config.bBlinkzeit; editable
rectangle at (497,401)-(660,434): text "Number of sequences"
rectangle at (667,442)-(744,474): text "%s * 600 ms"; shows DALI_Config.bBlinkdauer; invisible if DALI_Config.bActualFirmware < 7; editable
rectangle at (497,442)-(660,474): text "Duration of a sequence"; invisible if DALI_Config.bActualFirmware < 7
67 more shapes without text or variables
*)

(* Visualisation DALI 647/Private/visuGroupButton
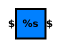
rectangle at (0,0)-(31,31): text "$Index$"; alarm colour if PrgDALIConfig.GroupConfig.axShortAddress[$Index$]
rectangle at (0,0)-(31,31): text "%s"; shows $Index$; invisible if NOT PrgDALIConfig.GroupConfig.axShortAddress[$Index$]; alarm colour if PrgDALIConfig.axGroupMember[$Index$]; toggles PrgDALIConfig.axGroupMember[$Index$]
*)

(* Visualisation Private/English/visuGroupSceneConfiguration
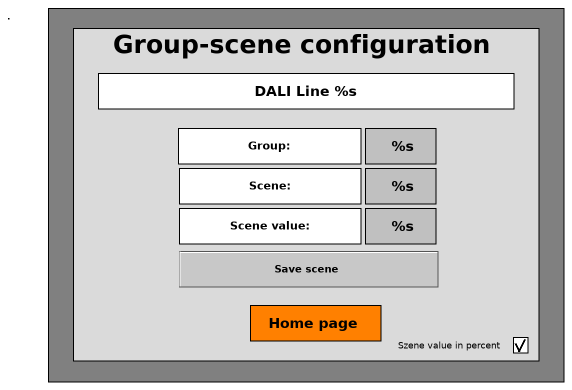
rectangle at (150,40)-(616,373): text "Group-scene configuration"
rounded rectangle at (327,317)-(458,353): text "Home page"; opens visuFrontPageDALI; tooltip Back to home page
rounded rectangle at (175,85)-(591,121): text "DALI Line %s"; shows DALI_Config.Dali_Linie; alarm colour if DALI_Config.keineJobliste; tooltip You can change the DALI Line only on the home page.
rectangle at (255,140)-(438,176): text "Group:"
rectangle at (442,140)-(513,176): text "%s"; shows DALI_Config.sGroup; tooltip Enter the number of the group (1 - 16); editable
button at (256,263)-(515,299): text "Save scene"; taps DALI_Config.sSaveScene; tooltip Save the configured dim levels in the ECGs.
rectangle at (256,180)-(438,216): text "Scene:"
rectangle at (442,180)-(513,216): text "%s"; shows DALI_Config.sScene; tooltip Select scene 1 - 16; editable
rectangle at (256,220)-(438,256): text "Scene value:"
rectangle at (442,220)-(513,256): text "%s"; shows DALI_Config.sSceneValue; tooltip Select scene 1 - 16; editable
rectangle at (473,346)-(589,369): text "Szene value in percent"
rectangle at (590,349)-(605,365): toggles DALI_Config.xDimmwertProzent
polyline at (592,351)-(602,363): invisible if NOT  DALI_Config.xDimmwertProzent; toggles DALI_Config.xDimmwertProzent
2 more shapes without text or variables
*)

(* Visualisation DALI 647/Private/visuIdentifyCurrentAddress
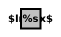
rectangle at (0,0)-(21,21): text "$Index$"; alarm colour if PrgDALIConfig.IdentifyControlGear.bCurrentShortAddress = $Index$; runs INTERN ASSIGN PrgDALIConfig.IdentifyControlGear.bCurrentShortAddress:=($Index$)
rectangle at (0,0)-(21,21): text "%s"; shows $Index$; invisible if PrgDALIConfig.IdentifyControlGear.axShortAddress[$Index$]
*)

(* Visualisation Private/English/visuLamp_status
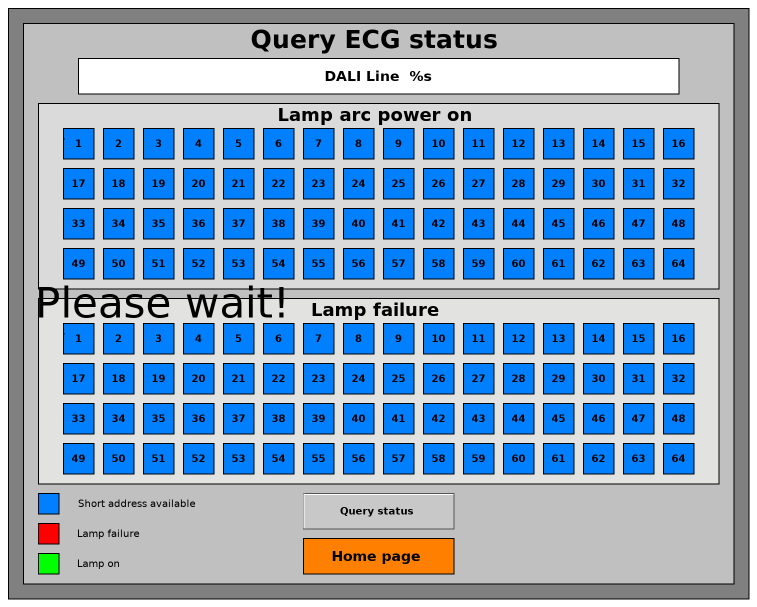
rectangle at (45,15)-(756,576): text "Query ECG status"
rounded rectangle at (325,530)-(476,566): text "Home page"; opens visuFrontPageDALI; tooltip Back to home page
rounded rectangle at (100,50)-(701,86): text "DALI Line  %s"; shows DALI_Config.Dali_Linie; alarm colour if DALI_Config.keineJobliste; tooltip You can change the DALI Line only on the home page.
rectangle at (60,95)-(741,281): text "Lamp arc power on"
rectangle at (85,120)-(116,151): text "1"; alarm colour if DALI_Config.Kurzadr[1]
rectangle at (85,120)-(116,151): text "1"; invisible if not DALI_Config.Kurzadr[1]; alarm colour if DALI_Config.LampeEin[1]
rectangle at (125,120)-(156,151): text "2"; alarm colour if DALI_Config.Kurzadr[2]
rectangle at (125,120)-(156,151): text "2"; invisible if not DALI_Config.Kurzadr[2]; alarm colour if DALI_Config.LampeEin[2]
rectangle at (165,120)-(196,151): text "3"; alarm colour if DALI_Config.Kurzadr[3]
rectangle at (165,120)-(196,151): text "3"; invisible if not DALI_Config.Kurzadr[3]; alarm colour if DALI_Config.LampeEin[3]
rectangle at (205,120)-(236,151): text "4"; alarm colour if DALI_Config.Kurzadr[4]
rectangle at (205,120)-(236,151): text "4"; invisible if not DALI_Config.Kurzadr[4]; alarm colour if DALI_Config.LampeEin[4]
rectangle at (245,120)-(276,151): text "5"; alarm colour if DALI_Config.Kurzadr[5]
rectangle at (245,120)-(276,151): text "5"; invisible if not DALI_Config.Kurzadr[5]; alarm colour if DALI_Config.LampeEin[5]
rectangle at (285,120)-(316,151): text "6"; alarm colour if DALI_Config.Kurzadr[6]
rectangle at (285,120)-(316,151): text "6"; invisible if not DALI_Config.Kurzadr[6]; alarm colour if DALI_Config.LampeEin[6]
rectangle at (325,120)-(356,151): text "7"; alarm colour if DALI_Config.Kurzadr[7]
rectangle at (325,120)-(356,151): text "7"; invisible if not DALI_Config.Kurzadr[7]; alarm colour if DALI_Config.LampeEin[7]
rectangle at (365,120)-(396,151): text "8"; alarm colour if DALI_Config.Kurzadr[8]
rectangle at (365,120)-(396,151): text "8"; invisible if not DALI_Config.Kurzadr[8]; alarm colour if DALI_Config.LampeEin[8]
rectangle at (405,120)-(436,151): text "9"; alarm colour if DALI_Config.Kurzadr[9]
rectangle at (405,120)-(436,151): text "9"; invisible if not DALI_Config.Kurzadr[9]; alarm colour if DALI_Config.LampeEin[9]
rectangle at (445,120)-(476,151): text "10"; alarm colour if DALI_Config.Kurzadr[10]
rectangle at (445,120)-(476,151): text "10"; invisible if not DALI_Config.Kurzadr[10]; alarm colour if DALI_Config.LampeEin[10]
rectangle at (485,120)-(516,151): text "11"; alarm colour if DALI_Config.Kurzadr[11]
rectangle at (485,120)-(516,151): text "11"; invisible if not DALI_Config.Kurzadr[11]; alarm colour if DALI_Config.LampeEin[11]
rectangle at (525,120)-(556,151): text "12"; alarm colour if DALI_Config.Kurzadr[12]
rectangle at (525,120)-(556,151): text "12"; invisible if not DALI_Config.Kurzadr[12]; alarm colour if DALI_Config.LampeEin[12]
rectangle at (565,120)-(596,151): text "13"; alarm colour if DALI_Config.Kurzadr[13]
rectangle at (565,120)-(596,151): text "13"; invisible if not DALI_Config.Kurzadr[13]; alarm colour if DALI_Config.LampeEin[13]
rectangle at (605,120)-(636,151): text "14"; alarm colour if DALI_Config.Kurzadr[14]
rectangle at (605,120)-(636,151): text "14"; invisible if not DALI_Config.Kurzadr[14]; alarm colour if DALI_Config.LampeEin[14]
rectangle at (645,120)-(676,151): text "15"; alarm colour if DALI_Config.Kurzadr[15]
rectangle at (645,120)-(676,151): text "15"; invisible if not DALI_Config.Kurzadr[15]; alarm colour if DALI_Config.LampeEin[15]
rectangle at (685,120)-(716,151): text "16"; alarm colour if DALI_Config.Kurzadr[16]
rectangle at (685,120)-(716,151): text "16"; invisible if not DALI_Config.Kurzadr[16]; alarm colour if DALI_Config.LampeEin[16]
rectangle at (85,160)-(116,191): text "17"; alarm colour if DALI_Config.Kurzadr[17]
rectangle at (85,160)-(116,191): text "17"; invisible if not DALI_Config.Kurzadr[17]; alarm colour if DALI_Config.LampeEin[17]
rectangle at (165,160)-(196,191): text "19"; alarm colour if DALI_Config.Kurzadr[19]
rectangle at (165,160)-(196,191): text "19"; invisible if not DALI_Config.Kurzadr[19]; alarm colour if DALI_Config.LampeEin[19]
rectangle at (125,160)-(156,191): text "18"; alarm colour if DALI_Config.Kurzadr[18]
rectangle at (125,160)-(156,191): text "18"; invisible if not DALI_Config.Kurzadr[18]; alarm colour if DALI_Config.LampeEin[18]
rectangle at (205,160)-(236,191): text "20"; alarm colour if DALI_Config.Kurzadr[20]
rectangle at (205,160)-(236,191): text "20"; invisible if not DALI_Config.Kurzadr[20]; alarm colour if DALI_Config.LampeEin[20]
rectangle at (245,160)-(276,191): text "21"; alarm colour if DALI_Config.Kurzadr[21]
rectangle at (245,160)-(276,191): text "21"; invisible if not DALI_Config.Kurzadr[21]; alarm colour if DALI_Config.LampeEin[21]
rectangle at (285,160)-(316,191): text "22"; alarm colour if DALI_Config.Kurzadr[22]
rectangle at (285,160)-(316,191): text "22"; invisible if not DALI_Config.Kurzadr[22]; alarm colour if DALI_Config.LampeEin[22]
rectangle at (325,160)-(356,191): text "23"; alarm colour if DALI_Config.Kurzadr[23]
rectangle at (325,160)-(356,191): text "23"; invisible if not DALI_Config.Kurzadr[23]; alarm colour if DALI_Config.LampeEin[23]
rectangle at (365,160)-(396,191): text "24"; alarm colour if DALI_Config.Kurzadr[24]
rectangle at (365,160)-(396,191): text "24"; invisible if not DALI_Config.Kurzadr[24]; alarm colour if DALI_Config.LampeEin[24]
rectangle at (405,160)-(436,191): text "25"; alarm colour if DALI_Config.Kurzadr[25]
rectangle at (405,160)-(436,191): text "25"; invisible if not DALI_Config.Kurzadr[25]; alarm colour if DALI_Config.LampeEin[25]
rectangle at (565,160)-(596,191): text "29"; alarm colour if DALI_Config.Kurzadr[29]
rectangle at (565,160)-(596,191): text "29"; invisible if not DALI_Config.Kurzadr[29]; alarm colour if DALI_Config.LampeEin[29]
rectangle at (525,160)-(556,191): text "28"; alarm colour if DALI_Config.Kurzadr[28]
rectangle at (525,160)-(556,191): text "28"; invisible if not DALI_Config.Kurzadr[28]; alarm colour if DALI_Config.LampeEin[28]
rectangle at (485,160)-(516,191): text "27"; alarm colour if DALI_Config.Kurzadr[27]
rectangle at (485,160)-(516,191): text "27"; invisible if not DALI_Config.Kurzadr[27]; alarm colour if DALI_Config.LampeEin[27]
rectangle at (445,160)-(476,191): text "26"; alarm colour if DALI_Config.Kurzadr[26]
rectangle at (445,160)-(476,191): text "26"; invisible if not DALI_Config.Kurzadr[26]; alarm colour if DALI_Config.LampeEin[26]
rectangle at (605,160)-(636,191): text "30"; alarm colour if DALI_Config.Kurzadr[30]
rectangle at (605,160)-(636,191): text "30"; invisible if not DALI_Config.Kurzadr[30]; alarm colour if DALI_Config.LampeEin[30]
rectangle at (645,160)-(676,191): text "31"; alarm colour if DALI_Config.Kurzadr[31]
rectangle at (645,160)-(676,191): text "31"; invisible if not DALI_Config.Kurzadr[31]; alarm colour if DALI_Config.LampeEin[31]
rectangle at (685,160)-(716,191): text "32"; alarm colour if DALI_Config.Kurzadr[32]
rectangle at (685,160)-(716,191): text "32"; invisible if not DALI_Config.Kurzadr[32]; alarm colour if DALI_Config.LampeEin[32]
rectangle at (85,200)-(116,231): text "33"; alarm colour if DALI_Config.Kurzadr[33]
rectangle at (85,200)-(116,231): text "33"; invisible if not DALI_Config.Kurzadr[33]; alarm colour if DALI_Config.LampeEin[33]
rectangle at (125,200)-(156,231): text "34"; alarm colour if DALI_Config.Kurzadr[34]
rectangle at (125,200)-(156,231): text "34"; invisible if not DALI_Config.Kurzadr[34]; alarm colour if DALI_Config.LampeEin[34]
rectangle at (205,200)-(236,231): text "36"; alarm colour if DALI_Config.Kurzadr[36]
rectangle at (205,200)-(236,231): text "36"; invisible if not DALI_Config.Kurzadr[36]; alarm colour if DALI_Config.LampeEin[36]
rectangle at (285,200)-(316,231): text "38"; alarm colour if DALI_Config.Kurzadr[38]
rectangle at (285,200)-(316,231): text "38"; invisible if not DALI_Config.Kurzadr[38]; alarm colour if DALI_Config.LampeEin[38]
rectangle at (325,200)-(356,231): text "39"; alarm colour if DALI_Config.Kurzadr[39]
rectangle at (325,200)-(356,231): text "39"; invisible if not DALI_Config.Kurzadr[39]; alarm colour if DALI_Config.LampeEin[39]
rectangle at (245,200)-(276,231): text "37"; alarm colour if DALI_Config.Kurzadr[37]
rectangle at (245,200)-(276,231): text "37"; invisible if not DALI_Config.Kurzadr[37]; alarm colour if DALI_Config.LampeEin[37]
rectangle at (165,200)-(196,231): text "35"; alarm colour if DALI_Config.Kurzadr[35]
rectangle at (165,200)-(196,231): text "35"; invisible if not DALI_Config.Kurzadr[35]; alarm colour if DALI_Config.LampeEin[35]
rectangle at (405,200)-(436,231): text "41"; alarm colour if DALI_Config.Kurzadr[41]
rectangle at (405,200)-(436,231): text "41"; invisible if not DALI_Config.Kurzadr[41]; alarm colour if DALI_Config.LampeEin[41]
rectangle at (445,200)-(476,231): text "42"; alarm colour if DALI_Config.Kurzadr[42]
rectangle at (445,200)-(476,231): text "42"; invisible if not DALI_Config.Kurzadr[42]; alarm colour if DALI_Config.LampeEin[42]
rectangle at (365,200)-(396,231): text "40"; alarm colour if DALI_Config.Kurzadr[40]
rectangle at (365,200)-(396,231): text "40"; invisible if not DALI_Config.Kurzadr[40]; alarm colour if DALI_Config.LampeEin[40]
rectangle at (485,200)-(516,231): text "43"; alarm colour if DALI_Config.Kurzadr[43]
rectangle at (485,200)-(516,231): text "43"; invisible if not DALI_Config.Kurzadr[43]; alarm colour if DALI_Config.LampeEin[43]
rectangle at (525,200)-(556,231): text "44"; alarm colour if DALI_Config.Kurzadr[44]
rectangle at (525,200)-(556,231): text "44"; invisible if not DALI_Config.Kurzadr[44]; alarm colour if DALI_Config.LampeEin[44]
rectangle at (565,200)-(596,231): text "45"; alarm colour if DALI_Config.Kurzadr[45]
rectangle at (565,200)-(596,231): text "45"; invisible if not DALI_Config.Kurzadr[45]; alarm colour if DALI_Config.LampeEin[45]
rectangle at (605,200)-(636,231): text "46"; alarm colour if DALI_Config.Kurzadr[46]
rectangle at (605,200)-(636,231): text "46"; invisible if not DALI_Config.Kurzadr[46]; alarm colour if DALI_Config.LampeEin[46]
rectangle at (645,200)-(676,231): text "47"; alarm colour if DALI_Config.Kurzadr[47]
rectangle at (645,200)-(676,231): text "47"; invisible if not DALI_Config.Kurzadr[47]; alarm colour if DALI_Config.LampeEin[47]
rectangle at (685,200)-(716,231): text "48"; alarm colour if DALI_Config.Kurzadr[48]
rectangle at (685,200)-(716,231): text "48"; invisible if not DALI_Config.Kurzadr[48]; alarm colour if DALI_Config.LampeEin[48]
rectangle at (85,240)-(116,271): text "49"; alarm colour if DALI_Config.Kurzadr[49]
rectangle at (85,240)-(116,271): text "49"; invisible if not DALI_Config.Kurzadr[49]; alarm colour if DALI_Config.LampeEin[49]
rectangle at (125,240)-(156,271): text "50"; alarm colour if DALI_Config.Kurzadr[50]
rectangle at (125,240)-(156,271): text "50"; invisible if not DALI_Config.Kurzadr[50]; alarm colour if DALI_Config.LampeEin[50]
rectangle at (165,240)-(196,271): text "51"; alarm colour if DALI_Config.Kurzadr[51]
rectangle at (165,240)-(196,271): text "51"; invisible if not DALI_Config.Kurzadr[51]; alarm colour if DALI_Config.LampeEin[51]
rectangle at (205,240)-(236,271): text "52"; alarm colour if DALI_Config.Kurzadr[52]
rectangle at (205,240)-(236,271): text "52"; invisible if not DALI_Config.Kurzadr[52]; alarm colour if DALI_Config.LampeEin[52]
rectangle at (245,240)-(276,271): text "53"; alarm colour if DALI_Config.Kurzadr[53]
rectangle at (245,240)-(276,271): text "53"; invisible if not DALI_Config.Kurzadr[53]; alarm colour if DALI_Config.LampeEin[53]
rectangle at (285,240)-(316,271): text "54"; alarm colour if DALI_Config.Kurzadr[54]
rectangle at (285,240)-(316,271): text "54"; invisible if not DALI_Config.Kurzadr[54]; alarm colour if DALI_Config.LampeEin[54]
rectangle at (325,240)-(356,271): text "55"; alarm colour if DALI_Config.Kurzadr[55]
rectangle at (325,240)-(356,271): text "55"; invisible if not DALI_Config.Kurzadr[55]; alarm colour if DALI_Config.LampeEin[55]
rectangle at (365,240)-(396,271): text "56"; alarm colour if DALI_Config.Kurzadr[56]
rectangle at (365,240)-(396,271): text "56"; invisible if not DALI_Config.Kurzadr[56]; alarm colour if DALI_Config.LampeEin[56]
rectangle at (405,240)-(436,271): text "57"; alarm colour if DALI_Config.Kurzadr[57]
rectangle at (405,240)-(436,271): text "57"; invisible if not DALI_Config.Kurzadr[57]; alarm colour if DALI_Config.LampeEin[57]
rectangle at (485,240)-(516,271): text "59"; alarm colour if DALI_Config.Kurzadr[59]
rectangle at (485,240)-(516,271): text "59"; invisible if not DALI_Config.Kurzadr[59]; alarm colour if DALI_Config.LampeEin[59]
rectangle at (525,240)-(556,271): text "60"; alarm colour if DALI_Config.Kurzadr[60]
rectangle at (525,240)-(556,271): text "60"; invisible if not DALI_Config.Kurzadr[60]; alarm colour if DALI_Config.LampeEin[60]
rectangle at (565,240)-(596,271): text "61"; alarm colour if DALI_Config.Kurzadr[61]
rectangle at (565,240)-(596,271): text "61"; invisible if not DALI_Config.Kurzadr[61]; alarm colour if DALI_Config.LampeEin[61]
rectangle at (605,240)-(636,271): text "62"; alarm colour if DALI_Config.Kurzadr[62]
rectangle at (605,240)-(636,271): text "62"; invisible if not DALI_Config.Kurzadr[62]; alarm colour if DALI_Config.LampeEin[62]
rectangle at (445,240)-(476,271): text "58"; alarm colour if DALI_Config.Kurzadr[58]
rectangle at (445,240)-(476,271): text "58"; invisible if not DALI_Config.Kurzadr[58]; alarm colour if DALI_Config.LampeEin[58]
rectangle at (645,240)-(676,271): text "63"; alarm colour if DALI_Config.Kurzadr[63]
rectangle at (645,240)-(676,271): text "63"; invisible if not DALI_Config.Kurzadr[63]; alarm colour if DALI_Config.LampeEin[63]
rectangle at (685,240)-(716,271): text "64"; alarm colour if DALI_Config.Kurzadr[64]
rectangle at (685,240)-(716,271): text "64"; invisible if not DALI_Config.Kurzadr[64]; alarm colour if DALI_Config.LampeEin[64]
rectangle at (60,290)-(741,476): text "Lamp failure"
rectangle at (85,315)-(116,346): text "1"; alarm colour if DALI_Config.Kurzadr[1]
rectangle at (85,315)-(116,346): text "1"; invisible if not DALI_Config.Kurzadr[1]; alarm colour if DALI_Config.Lampenausfall[1]
rectangle at (125,315)-(156,346): text "2"; alarm colour if DALI_Config.Kurzadr[2]
rectangle at (125,315)-(156,346): text "2"; invisible if not DALI_Config.Kurzadr[2]; alarm colour if DALI_Config.Lampenausfall[2]
rectangle at (165,315)-(196,346): text "3"; alarm colour if DALI_Config.Kurzadr[3]
rectangle at (165,315)-(196,346): text "3"; invisible if not DALI_Config.Kurzadr[3]; alarm colour if DALI_Config.Lampenausfall[3]
rectangle at (205,315)-(236,346): text "4"; alarm colour if DALI_Config.Kurzadr[4]
rectangle at (205,315)-(236,346): text "4"; invisible if not DALI_Config.Kurzadr[4]; alarm colour if DALI_Config.Lampenausfall[4]
rectangle at (245,315)-(276,346): text "5"; alarm colour if DALI_Config.Kurzadr[5]
rectangle at (245,315)-(276,346): text "5"; invisible if not DALI_Config.Kurzadr[5]; alarm colour if DALI_Config.Lampenausfall[5]
rectangle at (285,315)-(316,346): text "6"; alarm colour if DALI_Config.Kurzadr[6]
rectangle at (285,315)-(316,346): text "6"; invisible if not DALI_Config.Kurzadr[6]; alarm colour if DALI_Config.Lampenausfall[6]
rectangle at (325,315)-(356,346): text "7"; alarm colour if DALI_Config.Kurzadr[7]
rectangle at (325,315)-(356,346): text "7"; invisible if not DALI_Config.Kurzadr[7]; alarm colour if DALI_Config.Lampenausfall[7]
rectangle at (365,315)-(396,346): text "8"; alarm colour if DALI_Config.Kurzadr[8]
rectangle at (365,315)-(396,346): text "8"; invisible if not DALI_Config.Kurzadr[8]; alarm colour if DALI_Config.Lampenausfall[8]
rectangle at (405,315)-(436,346): text "9"; alarm colour if DALI_Config.Kurzadr[9]
rectangle at (405,315)-(436,346): text "9"; invisible if not DALI_Config.Kurzadr[9]; alarm colour if DALI_Config.Lampenausfall[9]
rectangle at (445,315)-(476,346): text "10"; alarm colour if DALI_Config.Kurzadr[10]
rectangle at (445,315)-(476,346): text "10"; invisible if not DALI_Config.Kurzadr[10]; alarm colour if DALI_Config.Lampenausfall[10]
rectangle at (485,315)-(516,346): text "11"; alarm colour if DALI_Config.Kurzadr[11]
rectangle at (485,315)-(516,346): text "11"; invisible if not DALI_Config.Kurzadr[11]; alarm colour if DALI_Config.Lampenausfall[11]
rectangle at (525,315)-(556,346): text "12"; alarm colour if DALI_Config.Kurzadr[12]
rectangle at (525,315)-(556,346): text "12"; invisible if not DALI_Config.Kurzadr[12]; alarm colour if DALI_Config.Lampenausfall[12]
rectangle at (565,315)-(596,346): text "13"; alarm colour if DALI_Config.Kurzadr[13]
rectangle at (565,315)-(596,346): text "13"; invisible if not DALI_Config.Kurzadr[13]; alarm colour if DALI_Config.Lampenausfall[13]
rectangle at (605,315)-(636,346): text "14"; alarm colour if DALI_Config.Kurzadr[14]
rectangle at (605,315)-(636,346): text "14"; invisible if not DALI_Config.Kurzadr[14]; alarm colour if DALI_Config.Lampenausfall[14]
rectangle at (645,315)-(676,346): text "15"; alarm colour if DALI_Config.Kurzadr[15]
rectangle at (645,315)-(676,346): text "15"; invisible if not DALI_Config.Kurzadr[15]; alarm colour if DALI_Config.Lampenausfall[15]
rectangle at (685,315)-(716,346): text "16"; alarm colour if DALI_Config.Kurzadr[16]
rectangle at (685,315)-(716,346): text "16"; invisible if not DALI_Config.Kurzadr[16]; alarm colour if DALI_Config.Lampenausfall[16]
rectangle at (85,355)-(116,386): text "17"; alarm colour if DALI_Config.Kurzadr[17]
rectangle at (85,355)-(116,386): text "17"; invisible if not DALI_Config.Kurzadr[17]; alarm colour if DALI_Config.Lampenausfall[17]
rectangle at (165,355)-(196,386): text "19"; alarm colour if DALI_Config.Kurzadr[19]
rectangle at (165,355)-(196,386): text "19"; invisible if not DALI_Config.Kurzadr[19]; alarm colour if DALI_Config.Lampenausfall[19]
rectangle at (125,355)-(156,386): text "18"; alarm colour if DALI_Config.Kurzadr[18]
rectangle at (125,355)-(156,386): text "18"; invisible if not DALI_Config.Kurzadr[18]; alarm colour if DALI_Config.Lampenausfall[18]
rectangle at (205,355)-(236,386): text "20"; alarm colour if DALI_Config.Kurzadr[20]
rectangle at (205,355)-(236,386): text "20"; invisible if not DALI_Config.Kurzadr[20]; alarm colour if DALI_Config.Lampenausfall[20]
rectangle at (245,355)-(276,386): text "21"; alarm colour if DALI_Config.Kurzadr[21]
rectangle at (245,355)-(276,386): text "21"; invisible if not DALI_Config.Kurzadr[21]; alarm colour if DALI_Config.Lampenausfall[21]
rectangle at (285,355)-(316,386): text "22"; alarm colour if DALI_Config.Kurzadr[22]
rectangle at (285,355)-(316,386): text "22"; invisible if not DALI_Config.Kurzadr[22]; alarm colour if DALI_Config.Lampenausfall[22]
rectangle at (325,355)-(356,386): text "23"; alarm colour if DALI_Config.Kurzadr[23]
rectangle at (325,355)-(356,386): text "23"; invisible if not DALI_Config.Kurzadr[23]; alarm colour if DALI_Config.Lampenausfall[23]
rectangle at (365,355)-(396,386): text "24"; alarm colour if DALI_Config.Kurzadr[24]
rectangle at (365,355)-(396,386): text "24"; invisible if not DALI_Config.Kurzadr[24]; alarm colour if DALI_Config.Lampenausfall[24]
rectangle at (405,355)-(436,386): text "25"; alarm colour if DALI_Config.Kurzadr[25]
rectangle at (405,355)-(436,386): text "25"; invisible if not DALI_Config.Kurzadr[25]; alarm colour if DALI_Config.Lampenausfall[25]
rectangle at (565,355)-(596,386): text "29"; alarm colour if DALI_Config.Kurzadr[29]
rectangle at (565,355)-(596,386): text "29"; invisible if not DALI_Config.Kurzadr[29]; alarm colour if DALI_Config.Lampenausfall[29]
rectangle at (525,355)-(556,386): text "28"; alarm colour if DALI_Config.Kurzadr[28]
rectangle at (525,355)-(556,386): text "28"; invisible if not DALI_Config.Kurzadr[28]; alarm colour if DALI_Config.Lampenausfall[28]
rectangle at (485,355)-(516,386): text "27"; alarm colour if DALI_Config.Kurzadr[27]
rectangle at (485,355)-(516,386): text "27"; invisible if not DALI_Config.Kurzadr[27]; alarm colour if DALI_Config.Lampenausfall[27]
rectangle at (445,355)-(476,386): text "26"; alarm colour if DALI_Config.Kurzadr[26]
rectangle at (445,355)-(476,386): text "26"; invisible if not DALI_Config.Kurzadr[26]; alarm colour if DALI_Config.Lampenausfall[26]
rectangle at (605,355)-(636,386): text "30"; alarm colour if DALI_Config.Kurzadr[30]
rectangle at (605,355)-(636,386): text "30"; invisible if not DALI_Config.Kurzadr[30]; alarm colour if DALI_Config.Lampenausfall[30]
rectangle at (645,355)-(676,386): text "31"; alarm colour if DALI_Config.Kurzadr[31]
rectangle at (645,355)-(676,386): text "31"; invisible if not DALI_Config.Kurzadr[31]; alarm colour if DALI_Config.Lampenausfall[31]
rectangle at (685,355)-(716,386): text "32"; alarm colour if DALI_Config.Kurzadr[32]
rectangle at (685,355)-(716,386): text "32"; invisible if not DALI_Config.Kurzadr[32]; alarm colour if DALI_Config.Lampenausfall[32]
rectangle at (85,395)-(116,426): text "33"; alarm colour if DALI_Config.Kurzadr[33]
rectangle at (85,395)-(116,426): text "33"; invisible if not DALI_Config.Kurzadr[33]; alarm colour if DALI_Config.Lampenausfall[33]
rectangle at (125,395)-(156,426): text "34"; alarm colour if DALI_Config.Kurzadr[34]
rectangle at (125,395)-(156,426): text "34"; invisible if not DALI_Config.Kurzadr[34]; alarm colour if DALI_Config.Lampenausfall[34]
rectangle at (205,395)-(236,426): text "36"; alarm colour if DALI_Config.Kurzadr[36]
rectangle at (205,395)-(236,426): text "36"; invisible if not DALI_Config.Kurzadr[36]; alarm colour if DALI_Config.Lampenausfall[36]
rectangle at (285,395)-(316,426): text "38"; alarm colour if DALI_Config.Kurzadr[38]
rectangle at (285,395)-(316,426): text "38"; invisible if not DALI_Config.Kurzadr[38]; alarm colour if DALI_Config.Lampenausfall[38]
rectangle at (325,395)-(356,426): text "39"; alarm colour if DALI_Config.Kurzadr[39]
rectangle at (325,395)-(356,426): text "39"; invisible if not DALI_Config.Kurzadr[39]; alarm colour if DALI_Config.Lampenausfall[39]
rectangle at (245,395)-(276,426): text "37"; alarm colour if DALI_Config.Kurzadr[37]
rectangle at (245,395)-(276,426): text "37"; invisible if not DALI_Config.Kurzadr[37]; alarm colour if DALI_Config.Lampenausfall[37]
rectangle at (165,395)-(196,426): text "35"; alarm colour if DALI_Config.Kurzadr[35]
rectangle at (165,395)-(196,426): text "35"; invisible if not DALI_Config.Kurzadr[35]; alarm colour if DALI_Config.Lampenausfall[35]
rectangle at (405,395)-(436,426): text "41"; alarm colour if DALI_Config.Kurzadr[41]
rectangle at (405,395)-(436,426): text "41"; invisible if not DALI_Config.Kurzadr[41]; alarm colour if DALI_Config.Lampenausfall[41]
rectangle at (445,395)-(476,426): text "42"; alarm colour if DALI_Config.Kurzadr[42]
rectangle at (445,395)-(476,426): text "42"; invisible if not DALI_Config.Kurzadr[42]; alarm colour if DALI_Config.Lampenausfall[42]
rectangle at (365,395)-(396,426): text "40"; alarm colour if DALI_Config.Kurzadr[40]
rectangle at (365,395)-(396,426): text "40"; invisible if not DALI_Config.Kurzadr[40]; alarm colour if DALI_Config.Lampenausfall[40]
rectangle at (485,395)-(516,426): text "43"; alarm colour if DALI_Config.Kurzadr[43]
rectangle at (485,395)-(516,426): text "43"; invisible if not DALI_Config.Kurzadr[43]; alarm colour if DALI_Config.Lampenausfall[43]
rectangle at (525,395)-(556,426): text "44"; alarm colour if DALI_Config.Kurzadr[44]
rectangle at (525,395)-(556,426): text "44"; invisible if not DALI_Config.Kurzadr[44]; alarm colour if DALI_Config.Lampenausfall[44]
rectangle at (565,395)-(596,426): text "45"; alarm colour if DALI_Config.Kurzadr[45]
rectangle at (565,395)-(596,426): text "45"; invisible if not DALI_Config.Kurzadr[45]; alarm colour if DALI_Config.Lampenausfall[45]
rectangle at (605,395)-(636,426): text "46"; alarm colour if DALI_Config.Kurzadr[46]
rectangle at (605,395)-(636,426): text "46"; invisible if not DALI_Config.Kurzadr[46]; alarm colour if DALI_Config.Lampenausfall[46]
rectangle at (645,395)-(676,426): text "47"; alarm colour if DALI_Config.Kurzadr[47]
rectangle at (645,395)-(676,426): text "47"; invisible if not DALI_Config.Kurzadr[47]; alarm colour if DALI_Config.Lampenausfall[47]
rectangle at (685,395)-(716,426): text "48"; alarm colour if DALI_Config.Kurzadr[48]
rectangle at (685,395)-(716,426): text "48"; invisible if not DALI_Config.Kurzadr[48]; alarm colour if DALI_Config.Lampenausfall[48]
rectangle at (85,435)-(116,466): text "49"; alarm colour if DALI_Config.Kurzadr[49]
rectangle at (85,435)-(116,466): text "49"; invisible if not DALI_Config.Kurzadr[49]; alarm colour if DALI_Config.Lampenausfall[49]
rectangle at (125,435)-(156,466): text "50"; alarm colour if DALI_Config.Kurzadr[50]
rectangle at (125,435)-(156,466): text "50"; invisible if not DALI_Config.Kurzadr[50]; alarm colour if DALI_Config.Lampenausfall[50]
rectangle at (165,435)-(196,466): text "51"; alarm colour if DALI_Config.Kurzadr[51]
rectangle at (165,435)-(196,466): text "51"; invisible if not DALI_Config.Kurzadr[51]; alarm colour if DALI_Config.Lampenausfall[51]
rectangle at (205,435)-(236,466): text "52"; alarm colour if DALI_Config.Kurzadr[52]
rectangle at (205,435)-(236,466): text "52"; invisible if not DALI_Config.Kurzadr[52]; alarm colour if DALI_Config.Lampenausfall[52]
rectangle at (245,435)-(276,466): text "53"; alarm colour if DALI_Config.Kurzadr[53]
rectangle at (245,435)-(276,466): text "53"; invisible if not DALI_Config.Kurzadr[53]; alarm colour if DALI_Config.Lampenausfall[53]
rectangle at (285,435)-(316,466): text "54"; alarm colour if DALI_Config.Kurzadr[54]
rectangle at (285,435)-(316,466): text "54"; invisible if not DALI_Config.Kurzadr[54]; alarm colour if DALI_Config.Lampenausfall[54]
rectangle at (325,435)-(356,466): text "55"; alarm colour if DALI_Config.Kurzadr[55]
rectangle at (325,435)-(356,466): text "55"; invisible if not DALI_Config.Kurzadr[55]; alarm colour if DALI_Config.Lampenausfall[55]
rectangle at (365,435)-(396,466): text "56"; alarm colour if DALI_Config.Kurzadr[56]
rectangle at (365,435)-(396,466): text "56"; invisible if not DALI_Config.Kurzadr[56]; alarm colour if DALI_Config.Lampenausfall[56]
rectangle at (405,435)-(436,466): text "57"; alarm colour if DALI_Config.Kurzadr[57]
rectangle at (405,435)-(436,466): text "57"; invisible if not DALI_Config.Kurzadr[57]; alarm colour if DALI_Config.Lampenausfall[57]
rectangle at (485,435)-(516,466): text "59"; alarm colour if DALI_Config.Kurzadr[59]
rectangle at (485,435)-(516,466): text "59"; invisible if not DALI_Config.Kurzadr[59]; alarm colour if DALI_Config.Lampenausfall[59]
rectangle at (525,435)-(556,466): text "60"; alarm colour if DALI_Config.Kurzadr[60]
rectangle at (525,435)-(556,466): text "60"; invisible if not DALI_Config.Kurzadr[60]; alarm colour if DALI_Config.Lampenausfall[60]
rectangle at (565,435)-(596,466): text "61"; alarm colour if DALI_Config.Kurzadr[61]
rectangle at (565,435)-(596,466): text "61"; invisible if not DALI_Config.Kurzadr[61]; alarm colour if DALI_Config.Lampenausfall[61]
rectangle at (605,435)-(636,466): text "62"; alarm colour if DALI_Config.Kurzadr[62]
rectangle at (605,435)-(636,466): text "62"; invisible if not DALI_Config.Kurzadr[62]; alarm colour if DALI_Config.Lampenausfall[62]
rectangle at (445,435)-(476,466): text "58"; alarm colour if DALI_Config.Kurzadr[58]
rectangle at (445,435)-(476,466): text "58"; invisible if not DALI_Config.Kurzadr[58]; alarm colour if DALI_Config.Lampenausfall[58]
rectangle at (645,435)-(676,466): text "63"; alarm colour if DALI_Config.Kurzadr[63]
rectangle at (645,435)-(676,466): text "63"; invisible if not DALI_Config.Kurzadr[63]; alarm colour if DALI_Config.Lampenausfall[63]
rectangle at (685,435)-(716,466): text "64"; alarm colour if DALI_Config.Kurzadr[64]
rectangle at (685,435)-(716,466): text "64"; invisible if not DALI_Config.Kurzadr[64]; alarm colour if DALI_Config.Lampenausfall[64]
button at (325,485)-(476,521): text "Query status"; taps DALI_Config.Status; tooltip If you click the button "Query Status", you will get the status "Lamp failure" and "Lamp arc power on" from the ECG.
rectangle at (98,485)-(259,506): text "Short address available"
rectangle at (97,515)-(228,536): text "Lamp failure"
rectangle at (97,545)-(168,566): text "Lamp on"
rectangle at (55,13)-(755,576): text "Please wait!"; invisible if NOT DALI_Config.mStatus
6 more shapes without text or variables
*)

(* Visualisation DALI 647/Private/visuNewShortAddress
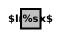
rectangle at (0,0)-(21,21): text "$Index$"; alarm colour if PrgDALIConfig.IdentifyControlGear.bNewShortAddress = $Index$; runs INTERN ASSIGN PrgDALIConfig.IdentifyControlGear.bNewShortAddress:=($Index$)
rectangle at (0,0)-(21,21): text "%s"; shows $Index$; invisible if PrgDALIConfig.IdentifyControlGear.axShortAddress[$Index$]; alarm colour if PrgDALIConfig.IdentifyControlGear.bNewShortAddress = $Index$; runs INTERN ASSIGN PrgDALIConfig.IdentifyControlGear.bNewShortAddress:=($Index$)
*)

(* Visualisation DALI 647/Private/visuOperatingHours
rectangle at (0,0)-(21,21): text "%s"; shows $Index$; alarm colour if PrgDALIConfig.axSelect[$Index$]; toggles PrgDALIConfig.axSelect[$Index$]
1 elements of other kinds (tables, trends, ...) not read
*)

(* Visualisation Private/English/visuScene_configuration
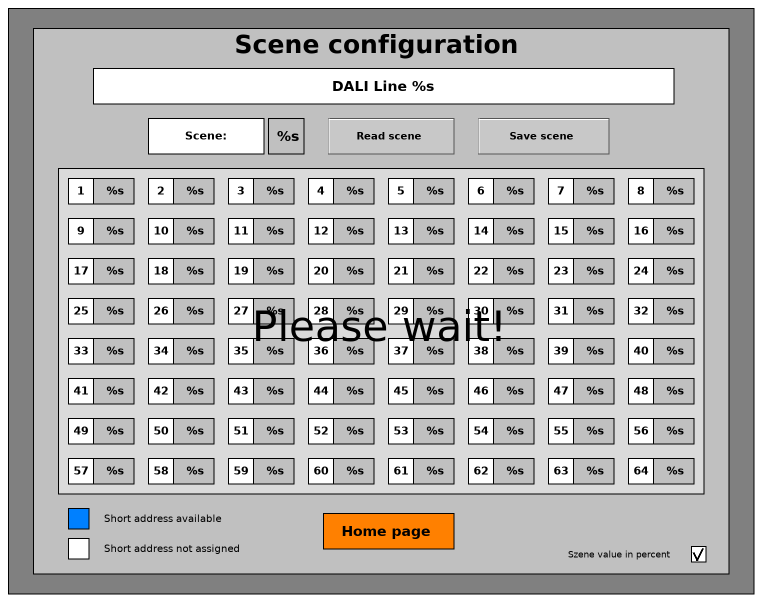
rectangle at (50,25)-(746,571): text "Scene configuration"
rounded rectangle at (340,510)-(471,546): text "Home page"; opens visuFrontPageDALI; tooltip Back to home page
rounded rectangle at (110,65)-(691,101): text "DALI Line %s"; shows DALI_Config.Dali_Linie; alarm colour if DALI_Config.keineJobliste; tooltip You can change the DALI Line only on the home page.
rectangle at (85,175)-(111,201): text "1"; alarm colour if Dali_Config.Kurzadr[1]
rectangle at (110,175)-(151,201): text "%s"; shows DALI_Config.Szenenwert[1]; tooltip 0 % = Off 1 - 100 % = Dim level 101 % = Mask; editable
button at (495,115)-(626,151): text "Save scene"; taps DALI_Config.SzeneSpeichern; tooltip Save the configured dim levels in the ECGs.
button at (345,115)-(471,151): text "Read scene"; taps DALI_Config.SzeneLesen; tooltip Read the saved scene values from the ECGs.
rectangle at (85,215)-(111,241): text "9"; alarm colour if Dali_Config.Kurzadr[9]
rectangle at (110,215)-(151,241): text "%s"; shows DALI_Config.Szenenwert[9]; tooltip 0 % = Off 1 - 100 % = Dim level 101 % = Mask; editable
rectangle at (85,255)-(111,281): text "17"; alarm colour if Dali_Config.Kurzadr[17]
rectangle at (110,255)-(151,281): text "%s"; shows DALI_Config.Szenenwert[17]; tooltip 0 % = Off 1 - 100 % = Dim level 101 % = Mask; editable
rectangle at (85,295)-(111,321): text "25"; alarm colour if Dali_Config.Kurzadr[25]
rectangle at (110,295)-(151,321): text "%s"; shows DALI_Config.Szenenwert[25]; tooltip 0 % = Off 1 - 100 % = Dim level 101 % = Mask; editable
rectangle at (85,335)-(111,361): text "33"; alarm colour if Dali_Config.Kurzadr[33]
rectangle at (110,335)-(151,361): text "%s"; shows DALI_Config.Szenenwert[33]; tooltip 0 % = Off 1 - 100 % = Dim level 101 % = Mask; editable
rectangle at (85,375)-(111,401): text "41"; alarm colour if Dali_Config.Kurzadr[41]
rectangle at (110,375)-(151,401): text "%s"; shows DALI_Config.Szenenwert[41]; tooltip 0 % = Off 1 - 100 % = Dim level 101 % = Mask; editable
rectangle at (85,415)-(111,441): text "49"; alarm colour if Dali_Config.Kurzadr[49]
rectangle at (110,415)-(151,441): text "%s"; shows DALI_Config.Szenenwert[49]; tooltip 0 % = Off 1 - 100 % = Dim level 101 % = Mask; editable
rectangle at (85,455)-(111,481): text "57"; alarm colour if Dali_Config.Kurzadr[57]
rectangle at (110,455)-(151,481): text "%s"; shows DALI_Config.Szenenwert[57]; tooltip 0 % = Off 1 - 100 % = Dim level 101 % = Mask; editable
rectangle at (165,175)-(191,201): text "2"; alarm colour if Dali_Config.Kurzadr[2]
rectangle at (190,175)-(231,201): text "%s"; shows DALI_Config.Szenenwert[2]; tooltip 0 % = Off 1 - 100 % = Dim level 101 % = Mask; editable
rectangle at (165,215)-(191,241): text "10"; alarm colour if Dali_Config.Kurzadr[10]
rectangle at (190,215)-(231,241): text "%s"; shows DALI_Config.Szenenwert[10]; tooltip 0 % = Off 1 - 100 % = Dim level 101 % = Mask; editable
rectangle at (165,255)-(191,281): text "18"; alarm colour if Dali_Config.Kurzadr[18]
rectangle at (190,255)-(231,281): text "%s"; shows DALI_Config.Szenenwert[18]; tooltip 0 % = Off 1 - 100 % = Dim level 101 % = Mask; editable
rectangle at (165,295)-(191,321): text "26"; alarm colour if Dali_Config.Kurzadr[26]
rectangle at (190,295)-(231,321): text "%s"; shows DALI_Config.Szenenwert[26]; tooltip 0 % = Off 1 - 100 % = Dim level 101 % = Mask; editable
rectangle at (165,335)-(191,361): text "34"; alarm colour if Dali_Config.Kurzadr[34]
rectangle at (190,335)-(231,361): text "%s"; shows DALI_Config.Szenenwert[34]; tooltip 0 % = Off 1 - 100 % = Dim level 101 % = Mask; editable
rectangle at (165,375)-(191,401): text "42"; alarm colour if Dali_Config.Kurzadr[42]
rectangle at (190,375)-(231,401): text "%s"; shows DALI_Config.Szenenwert[42]; tooltip 0 % = Off 1 - 100 % = Dim level 101 % = Mask; editable
rectangle at (165,415)-(191,441): text "50"; alarm colour if Dali_Config.Kurzadr[50]
rectangle at (190,415)-(231,441): text "%s"; shows DALI_Config.Szenenwert[50]; tooltip 0 % = Off 1 - 100 % = Dim level 101 % = Mask; editable
rectangle at (165,455)-(191,481): text "58"; alarm colour if Dali_Config.Kurzadr[58]
rectangle at (190,455)-(231,481): text "%s"; shows DALI_Config.Szenenwert[58]; tooltip 0 % = Off 1 - 100 % = Dim level 101 % = Mask; editable
rectangle at (245,175)-(271,201): text "3"; alarm colour if Dali_Config.Kurzadr[3]
rectangle at (270,175)-(311,201): text "%s"; shows DALI_Config.Szenenwert[3]; tooltip 0 % = Off 1 - 100 % = Dim level 101 % = Mask; editable
rectangle at (245,215)-(271,241): text "11"; alarm colour if Dali_Config.Kurzadr[11]
rectangle at (270,215)-(311,241): text "%s"; shows DALI_Config.Szenenwert[11]; tooltip 0 % = Off 1 - 100 % = Dim level 101 % = Mask; editable
rectangle at (245,255)-(271,281): text "19"; alarm colour if Dali_Config.Kurzadr[19]
rectangle at (270,255)-(311,281): text "%s"; shows DALI_Config.Szenenwert[19]; tooltip 0 % = Off 1 - 100 % = Dim level 101 % = Mask; editable
rectangle at (245,295)-(271,321): text "27"; alarm colour if Dali_Config.Kurzadr[27]
rectangle at (270,295)-(311,321): text "%s"; shows DALI_Config.Szenenwert[27]; tooltip 0 % = Off 1 - 100 % = Dim level 101 % = Mask; editable
rectangle at (245,335)-(271,361): text "35"; alarm colour if Dali_Config.Kurzadr[35]
rectangle at (270,335)-(311,361): text "%s"; shows DALI_Config.Szenenwert[35]; tooltip 0 % = Off 1 - 100 % = Dim level 101 % = Mask; editable
rectangle at (245,375)-(271,401): text "43"; alarm colour if Dali_Config.Kurzadr[43]
rectangle at (270,375)-(311,401): text "%s"; shows DALI_Config.Szenenwert[43]; tooltip 0 % = Off 1 - 100 % = Dim level 101 % = Mask; editable
rectangle at (245,415)-(271,441): text "51"; alarm colour if Dali_Config.Kurzadr[51]
rectangle at (270,415)-(311,441): text "%s"; shows DALI_Config.Szenenwert[51]; tooltip 0 % = Off 1 - 100 % = Dim level 101 % = Mask; editable
rectangle at (245,455)-(271,481): text "59"; alarm colour if Dali_Config.Kurzadr[59]
rectangle at (270,455)-(311,481): text "%s"; shows DALI_Config.Szenenwert[59]; tooltip 0 % = Off 1 - 100 % = Dim level 101 % = Mask; editable
rectangle at (325,175)-(351,201): text "4"; alarm colour if Dali_Config.Kurzadr[4]
rectangle at (350,175)-(391,201): text "%s"; shows DALI_Config.Szenenwert[4]; tooltip 0 % = Off 1 - 100 % = Dim level 101 % = Mask; editable
rectangle at (325,215)-(351,241): text "12"; alarm colour if Dali_Config.Kurzadr[12]
rectangle at (350,215)-(391,241): text "%s"; shows DALI_Config.Szenenwert[12]; tooltip 0 % = Off 1 - 100 % = Dim level 101 % = Mask; editable
rectangle at (325,255)-(351,281): text "20"; alarm colour if Dali_Config.Kurzadr[20]
rectangle at (350,255)-(391,281): text "%s"; shows DALI_Config.Szenenwert[20]; tooltip 0 % = Off 1 - 100 % = Dim level 101 % = Mask; editable
rectangle at (325,295)-(351,321): text "28"; alarm colour if Dali_Config.Kurzadr[28]
rectangle at (350,295)-(391,321): text "%s"; shows DALI_Config.Szenenwert[28]; tooltip 0 % = Off 1 - 100 % = Dim level 101 % = Mask; editable
rectangle at (325,335)-(351,361): text "36"; alarm colour if Dali_Config.Kurzadr[36]
rectangle at (350,335)-(391,361): text "%s"; shows DALI_Config.Szenenwert[36]; tooltip 0 % = Off 1 - 100 % = Dim level 101 % = Mask; editable
rectangle at (325,375)-(351,401): text "44"; alarm colour if Dali_Config.Kurzadr[44]
rectangle at (350,375)-(391,401): text "%s"; shows DALI_Config.Szenenwert[44]; tooltip 0 % = Off 1 - 100 % = Dim level 101 % = Mask; editable
rectangle at (325,415)-(351,441): text "52"; alarm colour if Dali_Config.Kurzadr[52]
rectangle at (350,415)-(391,441): text "%s"; shows DALI_Config.Szenenwert[52]; tooltip 0 % = Off 1 - 100 % = Dim level 101 % = Mask; editable
rectangle at (325,455)-(351,481): text "60"; alarm colour if Dali_Config.Kurzadr[60]
rectangle at (350,455)-(391,481): text "%s"; shows DALI_Config.Szenenwert[60]; tooltip 0 % = Off 1 - 100 % = Dim level 101 % = Mask; editable
rectangle at (405,175)-(431,201): text "5"; alarm colour if Dali_Config.Kurzadr[5]
rectangle at (430,175)-(471,201): text "%s"; shows DALI_Config.Szenenwert[5]; tooltip 0 % = Off 1 - 100 % = Dim level 101 % = Mask; editable
rectangle at (405,215)-(431,241): text "13"; alarm colour if Dali_Config.Kurzadr[13]
rectangle at (430,215)-(471,241): text "%s"; shows DALI_Config.Szenenwert[13]; tooltip 0 % = Off 1 - 100 % = Dim level 101 % = Mask; editable
rectangle at (405,255)-(431,281): text "21"; alarm colour if Dali_Config.Kurzadr[21]
rectangle at (430,255)-(471,281): text "%s"; shows DALI_Config.Szenenwert[21]; tooltip 0 % = Off 1 - 100 % = Dim level 101 % = Mask; editable
rectangle at (405,295)-(431,321): text "29"; alarm colour if Dali_Config.Kurzadr[29]
rectangle at (430,295)-(471,321): text "%s"; shows DALI_Config.Szenenwert[29]; tooltip 0 % = Off 1 - 100 % = Dim level 101 % = Mask; editable
rectangle at (405,335)-(431,361): text "37"; alarm colour if Dali_Config.Kurzadr[37]
rectangle at (430,335)-(471,361): text "%s"; shows DALI_Config.Szenenwert[37]; tooltip 0 % = Off 1 - 100 % = Dim level 101 % = Mask; editable
rectangle at (405,375)-(431,401): text "45"; alarm colour if Dali_Config.Kurzadr[45]
rectangle at (430,375)-(471,401): text "%s"; shows DALI_Config.Szenenwert[45]; tooltip 0 % = Off 1 - 100 % = Dim level 101 % = Mask; editable
rectangle at (405,415)-(431,441): text "53"; alarm colour if Dali_Config.Kurzadr[53]
rectangle at (430,415)-(471,441): text "%s"; shows DALI_Config.Szenenwert[53]; tooltip 0 % = Off 1 - 100 % = Dim level 101 % = Mask; editable
rectangle at (405,455)-(431,481): text "61"; alarm colour if Dali_Config.Kurzadr[61]
rectangle at (430,455)-(471,481): text "%s"; shows DALI_Config.Szenenwert[61]; tooltip 0 % = Off 1 - 100 % = Dim level 101 % = Mask; editable
rectangle at (485,175)-(511,201): text "6"; alarm colour if Dali_Config.Kurzadr[6]
rectangle at (510,175)-(551,201): text "%s"; shows DALI_Config.Szenenwert[6]; tooltip 0 % = Off 1 - 100 % = Dim level 101 % = Mask; editable
rectangle at (485,215)-(511,241): text "14"; alarm colour if Dali_Config.Kurzadr[14]
rectangle at (510,215)-(551,241): text "%s"; shows DALI_Config.Szenenwert[14]; tooltip 0 % = Off 1 - 100 % = Dim level 101 % = Mask; editable
rectangle at (485,255)-(511,281): text "22"; alarm colour if Dali_Config.Kurzadr[22]
rectangle at (510,255)-(551,281): text "%s"; shows DALI_Config.Szenenwert[22]; tooltip 0 % = Off 1 - 100 % = Dim level 101 % = Mask; editable
rectangle at (485,295)-(511,321): text "30"; alarm colour if Dali_Config.Kurzadr[30]
rectangle at (510,295)-(551,321): text "%s"; shows DALI_Config.Szenenwert[30]; tooltip 0 % = Off 1 - 100 % = Dim level 101 % = Mask; editable
rectangle at (485,335)-(511,361): text "38"; alarm colour if Dali_Config.Kurzadr[38]
rectangle at (510,335)-(551,361): text "%s"; shows DALI_Config.Szenenwert[38]; tooltip 0 % = Off 1 - 100 % = Dim level 101 % = Mask; editable
rectangle at (485,375)-(511,401): text "46"; alarm colour if Dali_Config.Kurzadr[46]
rectangle at (510,375)-(551,401): text "%s"; shows DALI_Config.Szenenwert[46]; tooltip 0 % = Off 1 - 100 % = Dim level 101 % = Mask; editable
rectangle at (485,415)-(511,441): text "54"; alarm colour if Dali_Config.Kurzadr[54]
rectangle at (510,415)-(551,441): text "%s"; shows DALI_Config.Szenenwert[54]; tooltip 0 % = Off 1 - 100 % = Dim level 101 % = Mask; editable
rectangle at (485,455)-(511,481): text "62"; alarm colour if Dali_Config.Kurzadr[62]
rectangle at (510,455)-(551,481): text "%s"; shows DALI_Config.Szenenwert[62]; tooltip 0 % = Off 1 - 100 % = Dim level 101 % = Mask; editable
rectangle at (565,175)-(591,201): text "7"; alarm colour if Dali_Config.Kurzadr[7]
rectangle at (590,175)-(631,201): text "%s"; shows DALI_Config.Szenenwert[7]; tooltip 0 % = Off 1 - 100 % = Dim level 101 % = Mask; editable
rectangle at (565,215)-(591,241): text "15"; alarm colour if Dali_Config.Kurzadr[15]
rectangle at (590,215)-(631,241): text "%s"; shows DALI_Config.Szenenwert[15]; tooltip 0 % = Off 1 - 100 % = Dim level 101 % = Mask; editable
rectangle at (565,255)-(591,281): text "23"; alarm colour if Dali_Config.Kurzadr[23]
rectangle at (590,255)-(631,281): text "%s"; shows DALI_Config.Szenenwert[23]; tooltip 0 % = Off 1 - 100 % = Dim level 101 % = Mask; editable
rectangle at (565,295)-(591,321): text "31"; alarm colour if Dali_Config.Kurzadr[31]
rectangle at (590,295)-(631,321): text "%s"; shows DALI_Config.Szenenwert[31]; tooltip 0 % = Off 1 - 100 % = Dim level 101 % = Mask; editable
rectangle at (565,335)-(591,361): text "39"; alarm colour if Dali_Config.Kurzadr[39]
rectangle at (590,335)-(631,361): text "%s"; shows DALI_Config.Szenenwert[39]; tooltip 0 % = Off 1 - 100 % = Dim level 101 % = Mask; editable
rectangle at (565,375)-(591,401): text "47"; alarm colour if Dali_Config.Kurzadr[47]
rectangle at (590,375)-(631,401): text "%s"; shows DALI_Config.Szenenwert[47]; tooltip 0 % = Off 1 - 100 % = Dim level 101 % = Mask; editable
rectangle at (565,415)-(591,441): text "55"; alarm colour if Dali_Config.Kurzadr[55]
rectangle at (590,415)-(631,441): text "%s"; shows DALI_Config.Szenenwert[55]; tooltip 0 % = Off 1 - 100 % = Dim level 101 % = Mask; editable
rectangle at (565,455)-(591,481): text "63"; alarm colour if Dali_Config.Kurzadr[63]
rectangle at (590,455)-(631,481): text "%s"; shows DALI_Config.Szenenwert[63]; tooltip 0 % = Off 1 - 100 % = Dim level 101 % = Mask; editable
rectangle at (645,175)-(671,201): text "8"; alarm colour if Dali_Config.Kurzadr[8]
rectangle at (670,175)-(711,201): text "%s"; shows DALI_Config.Szenenwert[8]; tooltip 0 % = Off 1 - 100 % = Dim level 101 % = Mask; editable
rectangle at (645,215)-(671,241): text "16"; alarm colour if Dali_Config.Kurzadr[16]
rectangle at (670,215)-(711,241): text "%s"; shows DALI_Config.Szenenwert[16]; tooltip 0 % = Off 1 - 100 % = Dim level 101 % = Mask; editable
rectangle at (645,255)-(671,281): text "24"; alarm colour if Dali_Config.Kurzadr[24]
rectangle at (670,255)-(711,281): text "%s"; shows DALI_Config.Szenenwert[24]; tooltip 0 % = Off 1 - 100 % = Dim level 101 % = Mask; editable
rectangle at (645,295)-(671,321): text "32"; alarm colour if Dali_Config.Kurzadr[32]
rectangle at (670,295)-(711,321): text "%s"; shows DALI_Config.Szenenwert[32]; tooltip 0 % = Off 1 - 100 % = Dim level 101 % = Mask; editable
rectangle at (645,335)-(671,361): text "40"; alarm colour if Dali_Config.Kurzadr[40]
rectangle at (670,335)-(711,361): text "%s"; shows DALI_Config.Szenenwert[40]; tooltip 0 % = Off 1 - 100 % = Dim level 101 % = Mask; editable
rectangle at (645,375)-(671,401): text "48"; alarm colour if Dali_Config.Kurzadr[48]
rectangle at (670,375)-(711,401): text "%s"; shows DALI_Config.Szenenwert[48]; tooltip 0 % = Off 1 - 100 % = Dim level 101 % = Mask; editable
rectangle at (645,415)-(671,441): text "56"; alarm colour if Dali_Config.Kurzadr[56]
rectangle at (670,415)-(711,441): text "%s"; shows DALI_Config.Szenenwert[56]; tooltip 0 % = Off 1 - 100 % = Dim level 101 % = Mask; editable
rectangle at (645,455)-(671,481): text "64"; alarm colour if Dali_Config.Kurzadr[64]
rectangle at (670,455)-(711,481): text "%s"; shows DALI_Config.Szenenwert[64]; tooltip 0 % = Off 1 - 100 % = Dim level 101 % = Mask; editable
rectangle at (165,115)-(281,151): text "Scene:"
rectangle at (285,115)-(321,151): text "%s"; shows DALI_Config.Szene; tooltip Select scene 1 - 16; editable
rectangle at (119,505)-(270,526): text "Short address available"
rectangle at (119,535)-(305,556): text "Short address not assigned"
rectangle at (51,78)-(742,568): text "Please wait!"; invisible if NOT DALI_Config.Unsichtbar
rectangle at (583,540)-(705,563): text "Szene value in percent"
rectangle at (708,543)-(723,559): toggles DALI_Config.xDimmwertProzent
polyline at (710,545)-(720,557): invisible if NOT  DALI_Config.xDimmwertProzent; toggles DALI_Config.xDimmwertProzent
4 more shapes without text or variables
*)

(* Visualisation DALI 647/Private/visuSceneValues
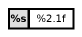
rectangle at (0,0)-(21,21): text "%s"; shows $Index$; alarm colour if PrgDALIConfig.SceneConfig.axShortAddress[$Index$]
rectangle at (20,0)-(66,21): text "%2.1f"; shows PrgDALIConfig.arSceneValues[$Index$]; editable
*)

